LIN {X 0,Y 224.704,Z 635.837,A -85,B 0,C 180,E1 -21459.979,E2 -21459.979} C_VEL
LIN {X 0,Y 218.18,Z 645.105,A -85,B 0,C 180,E1 -21463.55,E2 -21463.55} C_VEL
LIN {X 0,Y 212.599,Z 652.771,A -85,B 0,C 180,E1 -21467.337,E2 -21467.337} C_VEL
LIN {X 0,Y 208.284,Z 658.451,A -85,B 0,C 180,E1 -21470.904,E2 -21470.904} C_VEL
LIN {X 0,Y 204.923,Z 662.804,A -85,B 0,C 180,E1 -21474.336,E2 -21474.336} C_VEL
LIN {X 0,Y 201.755,Z 666.821,A -85,B 0,C 180,E1 -21478.499,E2 -21478.499} C_VEL
LIN {X 0,Y 199.518,Z 669.692,A -85,B 0,C 180,E1 -21482.746,E2 -21482.746} C_VEL
LIN {X 0,Y 197.956,Z 671.64,A -85,B 0,C 180,E1 -21487.383,E2 -21487.383} C_VEL
LIN {X 0,Y 197.23,Z 672.274,A -85,B 0,C 180,E1 -21491.294,E2 -21491.294} C_VEL
LIN {X 0,Y 196.985,Z 672.087,A -85,B 0,C 180,E1 -21495.537,E2 -21495.537} C_VEL
LIN {X 0,Y 196.96,Z 670.835,A -85,B 0,C 180,E1 -21499.722,E2 -21499.722} C_VEL
LIN {X 0,Y 197.621,Z 668.047,A -85,B 0,C 180,E1 -21504.738,E2 -21504.738} C_VEL
LIN {X 0,Y 198.077,Z 665.462,A -85,B 0,C 180,E1 -21507.966,E2 -21507.966} C_VEL
LIN {X 0,Y 199.268,Z 661.253,A -85,B 0,C 180,E1 -21512.021,E2 -21512.021} C_VEL
LIN {X 0,Y 201.021,Z 655.948,A -85,B 0,C 180,E1 -21516.02,E2 -21516.02} C_VEL
LIN {X 0,Y 203.624,Z 649.403,A -85,B 0,C 180,E1 -21519.937,E2 -21519.937} C_VEL
LIN {X 0,Y 206.969,Z 641.573,A -85,B 0,C 180,E1 -21523.75,E2 -21523.75} C_VEL
LIN {X 0,Y 211.157,Z 632.216,A -85,B 0,C 180,E1 -21527.43,E2 -21527.43} C_VEL
LIN {X 0,Y 215.924,Z 621.042,A -85,B 0,C 180,E1 -21530.979,E2 -21530.979} C_VEL
LIN {X 0,Y 220.656,Z 609.454,A -85,B 0,C 180,E1 -21533.959,E2 -21533.959} C_VEL
LIN {X 0,Y 225.409,Z 596.841,A -85,B 0,C 180,E1 -21536.628,E2 -21536.628} C_VEL
LIN {X 0,Y 230.179,Z 583.089,A -85,B 0,C 180,E1 -21538.993,E2 -21538.993} C_VEL
LIN {X 0,Y 234.489,Z 569.519,A -85,B 0,C 180,E1 -21540.881,E2 -21540.881} C_VEL
LIN {X 0,Y 238.368,Z 554.82,A -85,B 0,C 180,E1 -21542.553,E2 -21542.553} C_VEL
LIN {X 0,Y 241.83,Z 539.767,A -85,B 0,C 180,E1 -21543.891,E2 -21543.891} C_VEL
LIN {X 0,Y 244.962,Z 523.135,A -85,B 0,C 180,E1 -21545.016,E2 -21545.016} C_VEL
LIN {X 0,Y 247.354,Z 506.595,A -85,B 0,C 180,E1 -21545.812,E2 -21545.812} C_VEL
LIN {X 0,Y 248.927,Z 489.58,A -85,B 0,C 180,E1 -21546.363,E2 -21546.363} C_VEL
LIN {X 0,Y 255.202,Z 390.664,A -85,B 0,C 180,E1 -21548.897,E2 -21548.897} C_VEL
LIN {X 0,Y 247.991,Z 376.871,A -85,B 0,C 180,E1 -21551.304,E2 -21551.304} C_VEL
LIN {X 0,Y 240.547,Z 364.083,A -85,B 0,C 180,E1 -21554.004,E2 -21554.004} C_VEL
LIN {X 0,Y 233.352,Z 353.034,A -85,B 0,C 180,E1 -21556.877,E2 -21556.877} C_VEL
LIN {X 0,Y 227.132,Z 344.318,A -85,B 0,C 180,E1 -21559.64,E2 -21559.64} C_VEL
LIN {X 0,Y 224.214,Z 340.378,A -85,B 0,C 180,E1 -21561.054,E2 -21561.054} C_VEL
LIN {X 0,Y 220.981,Z 336.041,A -85,B 0,C 180,E1 -21562.732,E2 -21562.732} C_VEL
LIN {X 0,Y 217.624,Z 331.577,A -85,B 0,C 180,E1 -21564.617,E2 -21564.617} C_VEL
LIN {X 0,Y 214.933,Z 328.464,A -85,B 0,C 180,E1 -21566.228,E2 -21566.228} C_VEL
LIN {X 0,Y 213.999,Z 326.917,A -85,B 0,C 180,E1 -21566.854,E2 -21566.854} C_VEL
LIN {X 0,Y 211.261,Z 324.389,A -85,B 0,C 180,E1 -21568.646,E2 -21568.646} C_VEL
LIN {X 0,Y 209.46,Z 321.523,A -85,B 0,C 180,E1 -21570.03,E2 -21570.03} C_VEL
LIN {X 0,Y 206.617,Z 319.284,A -85,B 0,C 180,E1 -21572.205,E2 -21572.205} C_VEL
LIN {X 0,Y 205.081,Z 316.402,A -85,B 0,C 180,E1 -21573.68,E2 -21573.68} C_VEL
LIN {X 0,Y 204.71,Z 315.862,A -85,B 0,C 180,E1 -21574.04,E2 -21574.04} C_VEL
LIN {X 0,Y 201.778,Z 314.105,A -85,B 0,C 180,E1 -21576.883,E2 -21576.883} C_VEL
LIN {X 0,Y 200.084,Z 311.584,A -85,B 0,C 180,E1 -21579.031,E2 -21579.031} C_VEL
LIN {X 0,Y 199.696,Z 309.917,A -85,B 0,C 180,E1 -21579.796,E2 -21579.796} C_VEL
LIN {X 0,Y 199.771,Z 309.895,A -85,B 0,C 180,E1 -21583.653,E2 -21583.653} C_VEL
LIN {X 0,Y 199.871,Z 309.874,A -85,B 0,C 180,E1 -21587.819,E2 -21587.819} C_VEL
LIN {X 0,Y 200.086,Z 309.867,A -85,B 0,C 180,E1 -21591.922,E2 -21591.922} C_VEL
LIN {X 0,Y 200.315,Z 309.84,A -85,B 0,C 180,E1 -21597.988,E2 -21597.988} C_VEL
LIN {X 0,Y 200.476,Z 309.798,A -85,B 0,C 180,E1 -21599.999,E2 -21599.999} C_VEL
LIN {X 0,Y 200.026,Z 309.876,A -85,B 0,C 180,E1 -21604.028,E2 -21604.028} C_VEL
LIN {X 0,Y 200.061,Z 309.893,A -85,B 0,C 180,E1 -21607.315,E2 -21607.315} C_VEL
LIN {X 0,Y 200.946,Z 312.488,A -85,B 0,C 180,E1 -21608.674,E2 -21608.674} C_VEL
LIN {X 0,Y 203.236,Z 315.062,A -85,B 0,C 180,E1 -21611.215,E2 -21611.215} C_VEL
LIN {X 0,Y 205.117,Z 316.12,A -85,B 0,C 180,E1 -21612.93,E2 -21612.93} C_VEL
LIN {X 0,Y 206.498,Z 318.89,A -85,B 0,C 180,E1 -21614.284,E2 -21614.284} C_VEL
LIN {X 0,Y 208.777,Z 321.042,A -85,B 0,C 180,E1 -21616.097,E2 -21616.097} C_VEL
LIN {X 0,Y 209.862,Z 321.847,A -85,B 0,C 180,E1 -21616.88,E2 -21616.88} C_VEL
LIN {X 0,Y 210.233,Z 322.642,A -85,B 0,C 180,E1 -21617.184,E2 -21617.184} C_VEL
LIN {X 0,Y 212.25,Z 327.471,A -85,B 0,C 180,E1 -21618.802,E2 -21618.802} C_VEL
LIN {X 0,Y 216.82,Z 339.371,A -85,B 0,C 180,E1 -21622.139,E2 -21622.139} C_VEL
LIN {X 0,Y 218.895,Z 342.438,A -85,B 0,C 180,E1 -21623.347,E2 -21623.347} C_VEL
LIN {X 0,Y 224.048,Z 349.555,A -85,B 0,C 180,E1 -21626.049,E2 -21626.049} C_VEL
LIN {X 0,Y 231.097,Z 359.699,A -85,B 0,C 180,E1 -21629.302,E2 -21629.302} C_VEL
LIN {X 0,Y 235.181,Z 366.487,A -85,B 0,C 180,E1 -21631.045,E2 -21631.045} C_VEL
LIN {X 0,Y 240.195,Z 376.25,A -85,B 0,C 180,E1 -21633.083,E2 -21633.083} C_VEL
LIN {X 0,Y 245.695,Z 387.89,A -85,B 0,C 180,E1 -21635.177,E2 -21635.177} C_VEL
LIN {X 0,Y 250.053,Z 398.361,A -85,B 0,C 180,E1 -21636.771,E2 -21636.771} C_VEL
LIN {X 0,Y 242.749,Z 508.587,A -85,B 0,C 180,E1 -21639.663,E2 -21639.663} C_VEL
LIN {X 0,Y 240.64,Z 525.362,A -85,B 0,C 180,E1 -21640.335,E2 -21640.335} C_VEL
LIN {X 0,Y 237.748,Z 541.464,A -85,B 0,C 180,E1 -21641.241,E2 -21641.241} C_VEL
LIN {X 0,Y 234.346,Z 556.741,A -85,B 0,C 180,E1 -21642.396,E2 -21642.396} C_VEL
LIN {X 0,Y 230.362,Z 571.885,A -85,B 0,C 180,E1 -21643.883,E2 -21643.883} C_VEL
LIN {X 0,Y 225.648,Z 586.645,A -85,B 0,C 180,E1 -21645.694,E2 -21645.694} C_VEL
LIN {X 0,Y 220.975,Z 600.129,A -85,B 0,C 180,E1 -21647.789,E2 -21647.789} C_VEL
LIN {X 0,Y 216.272,Z 612.309,A -85,B 0,C 180,E1 -21650.074,E2 -21650.074} C_VEL
LIN {X 0,Y 211.517,Z 623.913,A -85,B 0,C 180,E1 -21652.732,E2 -21652.732} C_VEL
LIN {X 0,Y 206.703,Z 635.08,A -85,B 0,C 180,E1 -21655.875,E2 -21655.875} C_VEL
LIN {X 0,Y 202.378,Z 644.779,A -85,B 0,C 180,E1 -21659.188,E2 -21659.188} C_VEL
LIN {X 0,Y 198.341,Z 654.189,A -85,B 0,C 180,E1 -21663.142,E2 -21663.142} C_VEL
LIN {X 0,Y 194.763,Z 662.887,A -85,B 0,C 180,E1 -21667.735,E2 -21667.735} C_VEL
LIN {X 0,Y 192.402,Z 669.547,A -85,B 0,C 180,E1 -21672.22,E2 -21672.22} C_VEL
LIN {X 0,Y 191.102,Z 674.172,A -85,B 0,C 180,E1 -21676.17,E2 -21676.17} C_VEL
LIN {X 0,Y 190.231,Z 678.879,A -85,B 0,C 180,E1 -21681.502,E2 -21681.502} C_VEL
LIN {X 0,Y 190.191,Z 681.456,A -85,B 0,C 180,E1 -21685.762,E2 -21685.762} C_VEL
LIN {X 0,Y 190.296,Z 682.962,A -85,B 0,C 180,E1 -21690,E2 -21690} C_VEL
LIN {X 0,Y 190.133,Z 683.504,A -85,B 0,C 180,E1 -21694.24,E2 -21694.24} C_VEL
LIN {X 0,Y 190.218,Z 683.045,A -85,B 0,C 180,E1 -21698.499,E2 -21698.499} C_VEL
LIN {X 0,Y 190.881,Z 681.67,A -85,B 0,C 180,E1 -21702.763,E2 -21702.763} C_VEL
LIN {X 0,Y 192.373,Z 679.322,A -85,B 0,C 180,E1 -21706.994,E2 -21706.994} C_VEL
LIN {X 0,Y 194.698,Z 676.014,A -85,B 0,C 180,E1 -21711.16,E2 -21711.16} C_VEL
LIN {X 0,Y 197.894,Z 671.662,A -85,B 0,C 180,E1 -21715.225,E2 -21715.225} C_VEL
LIN {X 0,Y 201.988,Z 666.267,A -85,B 0,C 180,E1 -21719.152,E2 -21719.152} C_VEL
LIN {X 0,Y 207.01,Z 659.627,A -85,B 0,C 180,E1 -21722.902,E2 -21722.902} C_VEL
LIN {X 0,Y 213.655,Z 650.625,A -85,B 0,C 180,E1 -21726.893,E2 -21726.893} C_VEL
LIN {X 0,Y 220.364,Z 641.039,A -85,B 0,C 180,E1 -21730.228,E2 -21730.228} C_VEL
LIN {X 0,Y 227.8,Z 629.661,A -85,B 0,C 180,E1 -21733.35,E2 -21733.35} C_VEL
LIN {X 0,Y 234.942,Z 617.871,A -85,B 0,C 180,E1 -21735.884,E2 -21735.884} C_VEL
LIN {X 0,Y 241.451,Z 605.863,A -85,B 0,C 180,E1 -21737.975,E2 -21737.975} C_VEL
LIN {X 0,Y 248.161,Z 592.197,A -85,B 0,C 180,E1 -21739.876,E2 -21739.876} C_VEL
LIN {X 0,Y 254.139,Z 578.552,A -85,B 0,C 180,E1 -21741.374,E2 -21741.374} C_VEL
LIN {X 0,Y 259.557,Z 563.781,A -85,B 0,C 180,E1 -21742.692,E2 -21742.692} C_VEL
LIN {X 0,Y 264.238,Z 548.652,A -85,B 0,C 180,E1 -21743.729,E2 -21743.729} C_VEL
LIN {X 0,Y 268.405,Z 531.917,A -85,B 0,C 180,E1 -21744.591,E2 -21744.591} C_VEL
LIN {X 0,Y 271.417,Z 515.904,A -85,B 0,C 180,E1 -21745.177,E2 -21745.177} C_VEL
LIN {X 0,Y 273.367,Z 498.876,A -85,B 0,C 180,E1 -21745.66,E2 -21745.66} C_VEL
LIN {X 0,Y 279.986,Z 417.951,A -85,B 0,C 180,E1 -21747.514,E2 -21747.514} C_VEL
LIN {X 0,Y 275.543,Z 408.438,A -85,B 0,C 180,E1 -21749.967,E2 -21749.967} C_VEL
LIN {X 0,Y 271.529,Z 400.291,A -85,B 0,C 180,E1 -21752.452,E2 -21752.452} C_VEL
LIN {X 0,Y 266.969,Z 391.871,A -85,B 0,C 180,E1 -21755.707,E2 -21755.707} C_VEL
LIN {X 0,Y 263.419,Z 386.396,A -85,B 0,C 180,E1 -21758.705,E2 -21758.705} C_VEL
LIN {X 0,Y 260.513,Z 382.099,A -85,B 0,C 180,E1 -21761.74,E2 -21761.74} C_VEL
LIN {X 0,Y 258.214,Z 378.675,A -85,B 0,C 180,E1 -21764.965,E2 -21764.965} C_VEL
LIN {X 0,Y 257.777,Z 377.656,A -85,B 0,C 180,E1 -21765.797,E2 -21765.797} C_VEL
LIN {X 0,Y 255.553,Z 374.982,A -85,B 0,C 180,E1 -21773.018,E2 -21773.018} C_VEL
LIN {X 0,Y 256.078,Z 375.739,A -85,B 0,C 180,E1 -21777.641,E2 -21777.641} C_VEL
LIN {X 0,Y 258.062,Z 377.883,A -85,B 0,C 180,E1 -21782.12,E2 -21782.12} C_VEL
LIN {X 0,Y 260.464,Z 381.798,A -85,B 0,C 180,E1 -21785.614,E2 -21785.614} C_VEL
LIN {X 0,Y 261.202,Z 382.927,A -85,B 0,C 180,E1 -21786.47,E2 -21786.47} C_VEL
LIN {X 0,Y 264.003,Z 387.156,A -85,B 0,C 180,E1 -21789.264,E2 -21789.264} C_VEL
LIN {X 0,Y 267.122,Z 392.052,A -85,B 0,C 180,E1 -21791.85,E2 -21791.85} C_VEL
LIN {X 0,Y 271.202,Z 398.501,A -85,B 0,C 180,E1 -21794.696,E2 -21794.696} C_VEL
LIN {X 0,Y 276.177,Z 406.975,A -85,B 0,C 180,E1 -21797.674,E2 -21797.674} C_VEL
LIN {X 0,Y 280.247,Z 414.31,A -85,B 0,C 180,E1 -21799.832,E2 -21799.832} C_VEL
LIN {X 0,Y 273.006,Z 500.411,A -85,B 0,C 180,E1 -21801.818,E2 -21801.818} C_VEL
LIN {X 0,Y 270.274,Z 517.579,A -85,B 0,C 180,E1 -21802.37,E2 -21802.37} C_VEL
LIN {X 0,Y 266.884,Z 533.687,A -85,B 0,C 180,E1 -21803.19,E2 -21803.19} C_VEL
LIN {X 0,Y 262.691,Z 548.993,A -85,B 0,C 180,E1 -21804.19,E2 -21804.19} C_VEL
LIN {X 0,Y 257.769,Z 563.8,A -85,B 0,C 180,E1 -21805.425,E2 -21805.425} C_VEL
LIN {X 0,Y 252.193,Z 577.919,A -85,B 0,C 180,E1 -21806.904,E2 -21806.904} C_VEL
LIN {X 0,Y 245.781,Z 591.955,A -85,B 0,C 180,E1 -21808.756,E2 -21808.756} C_VEL
LIN {X 0,Y 239.278,Z 604.411,A -85,B 0,C 180,E1 -21810.782,E2 -21810.782} C_VEL
LIN {X 0,Y 232.265,Z 616.607,A -85,B 0,C 180,E1 -21813.266,E2 -21813.266} C_VEL
LIN {X 0,Y 225.616,Z 627.114,A -85,B 0,C 180,E1 -21815.913,E2 -21815.913} C_VEL
LIN {X 0,Y 219.013,Z 636.625,A -85,B 0,C 180,E1 -21818.906,E2 -21818.906} C_VEL
LIN {X 0,Y 212.212,Z 645.786,A -85,B 0,C 180,E1 -21822.534,E2 -21822.534} C_VEL
LIN {X 0,Y 206.881,Z 652.722,A -85,B 0,C 180,E1 -21826.022,E2 -21826.022} C_VEL
LIN {X 0,Y 201.943,Z 658.863,A -85,B 0,C 180,E1 -21829.966,E2 -21829.966} C_VEL
LIN {X 0,Y 197.855,Z 663.805,A -85,B 0,C 180,E1 -21834.121,E2 -21834.121} C_VEL
LIN {X 0,Y 195.325,Z 666.777,A -85,B 0,C 180,E1 -21837.335,E2 -21837.335} C_VEL
LIN {X 0,Y 192.83,Z 669.746,A -85,B 0,C 180,E1 -21841.718,E2 -21841.718} C_VEL
LIN {X 0,Y 191.144,Z 671.643,A -85,B 0,C 180,E1 -21846.143,E2 -21846.143} C_VEL
LIN {X 0,Y 190.213,Z 672.467,A -85,B 0,C 180,E1 -21850.577,E2 -21850.577} C_VEL
LIN {X 0,Y 189.912,Z 672.341,A -85,B 0,C 180,E1 -21854.986,E2 -21854.986} C_VEL
LIN {X 0,Y 189.838,Z 671.158,A -85,B 0,C 180,E1 -21859.332,E2 -21859.332} C_VEL
LIN {X 0,Y 190.282,Z 669.078,A -85,B 0,C 180,E1 -21863.638,E2 -21863.638} C_VEL
LIN {X 0,Y 190.973,Z 665.916,A -85,B 0,C 180,E1 -21867.891,E2 -21867.891} C_VEL
LIN {X 0,Y 192.18,Z 661.802,A -85,B 0,C 180,E1 -21872.096,E2 -21872.096} C_VEL
LIN {X 0,Y 193.97,Z 656.546,A -85,B 0,C 180,E1 -21876.24,E2 -21876.24} C_VEL
LIN {X 0,Y 196.647,Z 650.108,A -85,B 0,C 180,E1 -21880.294,E2 -21880.294} C_VEL
LIN {X 0,Y 200.106,Z 642.393,A -85,B 0,C 180,E1 -21884.232,E2 -21884.232} C_VEL
LIN {X 0,Y 204.419,Z 633.103,A -85,B 0,C 180,E1 -21888.024,E2 -21888.024} C_VEL
LIN {X 0,Y 208.705,Z 623.53,A -85,B 0,C 180,E1 -21891.223,E2 -21891.223} C_VEL
LIN {X 0,Y 213.549,Z 612.39,A -85,B 0,C 180,E1 -21894.291,E2 -21894.291} C_VEL
LIN {X 0,Y 218.336,Z 600.324,A -85,B 0,C 180,E1 -21897.043,E2 -21897.043} C_VEL
LIN {X 0,Y 223.623,Z 585.949,A -85,B 0,C 180,E1 -21899.669,E2 -21899.669} C_VEL
LIN {X 0,Y 228.502,Z 571.289,A -85,B 0,C 180,E1 -21901.783,E2 -21901.783} C_VEL
LIN {X 0,Y 232.522,Z 556.903,A -85,B 0,C 180,E1 -21903.477,E2 -21903.477} C_VEL
LIN {X 0,Y 236.289,Z 541.265,A -85,B 0,C 180,E1 -21904.929,E2 -21904.929} C_VEL
LIN {X 0,Y 239.548,Z 525.061,A -85,B 0,C 180,E1 -21906.058,E2 -21906.058} C_VEL
LIN {X 0,Y 241.952,Z 509.331,A -85,B 0,C 180,E1 -21906.87,E2 -21906.87} C_VEL
LIN {X 0,Y 243.738,Z 491.917,A -85,B 0,C 180,E1 -21907.458,E2 -21907.458} C_VEL
LIN {X 0,Y 250.218,Z 393.361,A -85,B 0,C 180,E1 -21910.013,E2 -21910.013} C_VEL
LIN {X 0,Y 243.332,Z 380.216,A -85,B 0,C 180,E1 -21912.435,E2 -21912.435} C_VEL
LIN {X 0,Y 236.792,Z 368.826,A -85,B 0,C 180,E1 -21914.936,E2 -21914.936} C_VEL
LIN {X 0,Y 230.444,Z 358.854,A -85,B 0,C 180,E1 -21917.587,E2 -21917.587} C_VEL
LIN {X 0,Y 224.274,Z 350.024,A -85,B 0,C 180,E1 -21920.446,E2 -21920.446} C_VEL
LIN {X 0,Y 221.012,Z 345.557,A -85,B 0,C 180,E1 -21922.106,E2 -21922.106} C_VEL
LIN {X 0,Y 218.342,Z 341.865,A -85,B 0,C 180,E1 -21923.567,E2 -21923.567} C_VEL
LIN {X 0,Y 215.202,Z 337.669,A -85,B 0,C 180,E1 -21925.411,E2 -21925.411} C_VEL
LIN {X 0,Y 212.429,Z 334.12,A -85,B 0,C 180,E1 -21927.178,E2 -21927.178} C_VEL
LIN {X 0,Y 210.816,Z 332.472,A -85,B 0,C 180,E1 -21928.25,E2 -21928.25} C_VEL
LIN {X 0,Y 208.297,Z 329.149,A -85,B 0,C 180,E1 -21930.119,E2 -21930.119} C_VEL
LIN {X 0,Y 207.591,Z 328.144,A -85,B 0,C 180,E1 -21930.681,E2 -21930.681} C_VEL
LIN {X 0,Y 204.877,Z 325.744,A -85,B 0,C 180,E1 -21932.871,E2 -21932.871} C_VEL
LIN {X 0,Y 203.357,Z 322.849,A -85,B 0,C 180,E1 -21934.404,E2 -21934.404} C_VEL
LIN {X 0,Y 200.049,Z 320.467,A -85,B 0,C 180,E1 -21937.81,E2 -21937.81} C_VEL
LIN {X 0,Y 198.536,Z 317.752,A -85,B 0,C 180,E1 -21939.943,E2 -21939.943} C_VEL
LIN {X 0,Y 198.159,Z 316.828,A -85,B 0,C 180,E1 -21940.578,E2 -21940.578} C_VEL
LIN {X 0,Y 194.367,Z 314.325,A -85,B 0,C 180,E1 -21948.528,E2 -21948.528} C_VEL
LIN {X 0,Y 193.907,Z 313.392,A -85,B 0,C 180,E1 -21951.663,E2 -21951.663} C_VEL
LIN {X 0,Y 194.521,Z 313.913,A -85,B 0,C 180,E1 -21958.446,E2 -21958.446} C_VEL
LIN {X 0,Y 195.475,Z 314.975,A -85,B 0,C 180,E1 -21961.286,E2 -21961.286} C_VEL
LIN {X 0,Y 197.619,Z 316.548,A -85,B 0,C 180,E1 -21965.271,E2 -21965.271} C_VEL
LIN {X 0,Y 198.722,Z 316.968,A -85,B 0,C 180,E1 -21966.79,E2 -21966.79} C_VEL
LIN {X 0,Y 199.805,Z 319.573,A -85,B 0,C 180,E1 -21968.426,E2 -21968.426} C_VEL
LIN {X 0,Y 202.055,Z 322.006,A -85,B 0,C 180,E1 -21970.964,E2 -21970.964} C_VEL
LIN {X 0,Y 203.513,Z 322.95,A -85,B 0,C 180,E1 -21972.349,E2 -21972.349} C_VEL
LIN {X 0,Y 205.331,Z 326.072,A -85,B 0,C 180,E1 -21974.122,E2 -21974.122} C_VEL
LIN {X 0,Y 208.079,Z 328.6,A -85,B 0,C 180,E1 -21976.309,E2 -21976.309} C_VEL
LIN {X 0,Y 210.43,Z 332.062,A -85,B 0,C 180,E1 -21978.096,E2 -21978.096} C_VEL
LIN {X 0,Y 212.297,Z 333.845,A -85,B 0,C 180,E1 -21979.331,E2 -21979.331} C_VEL
LIN {X 0,Y 214.989,Z 337.505,A -85,B 0,C 180,E1 -21981.074,E2 -21981.074} C_VEL
LIN {X 0,Y 216.463,Z 339.261,A -85,B 0,C 180,E1 -21981.954,E2 -21981.954} C_VEL
LIN {X 0,Y 218.895,Z 342.438,A -85,B 0,C 180,E1 -21983.347,E2 -21983.347} C_VEL
LIN {X 0,Y 220.304,Z 344.535,A -85,B 0,C 180,E1 -21984.13,E2 -21984.13} C_VEL
LIN {X 0,Y 221.475,Z 347.199,A -85,B 0,C 180,E1 -21984.818,E2 -21984.818} C_VEL
LIN {X 0,Y 225.862,Z 361.333,A -85,B 0,C 180,E1 -21987.461,E2 -21987.461} C_VEL
LIN {X 0,Y 228.001,Z 365.171,A -85,B 0,C 180,E1 -21988.481,E2 -21988.481} C_VEL
LIN {X 0,Y 231.897,Z 371.817,A -85,B 0,C 180,E1 -21990.222,E2 -21990.222} C_VEL
LIN {X 0,Y 236.874,Z 381.772,A -85,B 0,C 180,E1 -21992.342,E2 -21992.342} C_VEL
LIN {X 0,Y 242.247,Z 393.639,A -85,B 0,C 180,E1 -21994.483,E2 -21994.483} C_VEL
LIN {X 0,Y 245.234,Z 400.816,A -85,B 0,C 180,E1 -21995.625,E2 -21995.625} C_VEL
LIN {X 0,Y 237.721,Z 509.196,A -85,B 0,C 180,E1 -21998.478,E2 -21998.478} C_VEL
LIN {X 0,Y 235.469,Z 526.323,A -85,B 0,C 180,E1 -21999.188,E2 -21999.188} C_VEL
LIN {X 0,Y 232.505,Z 541.938,A -85,B 0,C 180,E1 -22000.082,E2 -22000.082} C_VEL
LIN {X 0,Y 228.731,Z 558.063,A -85,B 0,C 180,E1 -22001.335,E2 -22001.335} C_VEL
LIN {X 0,Y 224.903,Z 572.108,A -85,B 0,C 180,E1 -22002.748,E2 -22002.748} C_VEL
LIN {X 0,Y 220.172,Z 586.443,A -85,B 0,C 180,E1 -22004.529,E2 -22004.529} C_VEL
LIN {X 0,Y 215.218,Z 600.232,A -85,B 0,C 180,E1 -22006.705,E2 -22006.705} C_VEL
LIN {X 0,Y 209.912,Z 613.358,A -85,B 0,C 180,E1 -22009.242,E2 -22009.242} C_VEL
LIN {X 0,Y 204.673,Z 625.551,A -85,B 0,C 180,E1 -22012.162,E2 -22012.162} C_VEL
LIN {X 0,Y 200.055,Z 635.84,A -85,B 0,C 180,E1 -22015.19,E2 -22015.19} C_VEL
LIN {X 0,Y 195.587,Z 645.376,A -85,B 0,C 180,E1 -22018.599,E2 -22018.599} C_VEL
LIN {X 0,Y 191.416,Z 654.642,A -85,B 0,C 180,E1 -22022.681,E2 -22022.681} C_VEL
LIN {X 0,Y 188.087,Z 662.381,A -85,B 0,C 180,E1 -22026.9,E2 -22026.9} C_VEL
LIN {X 0,Y 185.758,Z 668.434,A -85,B 0,C 180,E1 -22031.056,E2 -22031.056} C_VEL
LIN {X 0,Y 184.142,Z 673.77,A -85,B 0,C 180,E1 -22035.636,E2 -22035.636} C_VEL
LIN {X 0,Y 183.162,Z 678.54,A -85,B 0,C 180,E1 -22041.172,E2 -22041.172} C_VEL
LIN {X 0,Y 183.111,Z 681.148,A -85,B 0,C 180,E1 -22045.598,E2 -22045.598} C_VEL
LIN {X 0,Y 183.199,Z 682.712,A -85,B 0,C 180,E1 -22050,E2 -22050} C_VEL
LIN {X 0,Y 183.029,Z 683.281,A -85,B 0,C 180,E1 -22054.405,E2 -22054.405} C_VEL
LIN {X 0,Y 183.159,Z 682.879,A -85,B 0,C 180,E1 -22058.829,E2 -22058.829} C_VEL
LIN {X 0,Y 183.889,Z 681.531,A -85,B 0,C 180,E1 -22063.257,E2 -22063.257} C_VEL
LIN {X 0,Y 185.517,Z 679.244,A -85,B 0,C 180,E1 -22067.642,E2 -22067.642} C_VEL
LIN {X 0,Y 188.002,Z 675.97,A -85,B 0,C 180,E1 -22071.952,E2 -22071.952} C_VEL
LIN {X 0,Y 191.407,Z 671.682,A -85,B 0,C 180,E1 -22076.143,E2 -22076.143} C_VEL
LIN {X 0,Y 195.737,Z 666.321,A -85,B 0,C 180,E1 -22080.177,E2 -22080.177} C_VEL
LIN {X 0,Y 201.036,Z 659.752,A -85,B 0,C 180,E1 -22084.011,E2 -22084.011} C_VEL
LIN {X 0,Y 207.991,Z 650.829,A -85,B 0,C 180,E1 -22088.073,E2 -22088.073} C_VEL
LIN {X 0,Y 214.961,Z 641.341,A -85,B 0,C 180,E1 -22091.457,E2 -22091.457} C_VEL
LIN {X 0,Y 222.676,Z 630.062,A -85,B 0,C 180,E1 -22094.608,E2 -22094.608} C_VEL
LIN {X 0,Y 230.066,Z 618.339,A -85,B 0,C 180,E1 -22097.151,E2 -22097.151} C_VEL
LIN {X 0,Y 237.263,Z 605.581,A -85,B 0,C 180,E1 -22099.381,E2 -22099.381} C_VEL
LIN {X 0,Y 244.312,Z 591.685,A -85,B 0,C 180,E1 -22101.288,E2 -22101.288} C_VEL
LIN {X 0,Y 250.409,Z 577.981,A -85,B 0,C 180,E1 -22102.786,E2 -22102.786} C_VEL
LIN {X 0,Y 255.983,Z 563.171,A -85,B 0,C 180,E1 -22104.089,E2 -22104.089} C_VEL
LIN {X 0,Y 260.819,Z 547.936,A -85,B 0,C 180,E1 -22105.102,E2 -22105.102} C_VEL
LIN {X 0,Y 264.973,Z 531.469,A -85,B 0,C 180,E1 -22105.941,E2 -22105.941} C_VEL
LIN {X 0,Y 268.089,Z 515.106,A -85,B 0,C 180,E1 -22106.525,E2 -22106.525} C_VEL
LIN {X 0,Y 270.033,Z 498.486,A -85,B 0,C 180,E1 -22106.988,E2 -22106.988} C_VEL
LIN {X 0,Y 276.521,Z 421.533,A -85,B 0,C 180,E1 -22108.743,E2 -22108.743} C_VEL
LIN {X 0,Y 272.814,Z 413.288,A -85,B 0,C 180,E1 -22110.935,E2 -22110.935} C_VEL
LIN {X 0,Y 269.158,Z 405.674,A -85,B 0,C 180,E1 -22113.335,E2 -22113.335} C_VEL
LIN {X 0,Y 264.696,Z 397.181,A -85,B 0,C 180,E1 -22116.749,E2 -22116.749} C_VEL
LIN {X 0,Y 261.859,Z 392.902,A -85,B 0,C 180,E1 -22119.285,E2 -22119.285} C_VEL
LIN {X 0,Y 259.2,Z 388.803,A -85,B 0,C 180,E1 -22122.219,E2 -22122.219} C_VEL
LIN {X 0,Y 257.029,Z 385.312,A -85,B 0,C 180,E1 -22125.468,E2 -22125.468} C_VEL
LIN {X 0,Y 256.69,Z 384.609,A -85,B 0,C 180,E1 -22126.134,E2 -22126.134} C_VEL
LIN {X 0,Y 254.678,Z 382.039,A -85,B 0,C 180,E1 -22132.994,E2 -22132.994} C_VEL
LIN {X 0,Y 255.195,Z 382.804,A -85,B 0,C 180,E1 -22137.633,E2 -22137.633} C_VEL
LIN {X 0,Y 257.006,Z 384.816,A -85,B 0,C 180,E1 -22141.848,E2 -22141.848} C_VEL
LIN {X 0,Y 259.246,Z 388.619,A -85,B 0,C 180,E1 -22145.25,E2 -22145.25} C_VEL
LIN {X 0,Y 259.932,Z 389.743,A -85,B 0,C 180,E1 -22146.088,E2 -22146.088} C_VEL
LIN {X 0,Y 262.662,Z 393.994,A -85,B 0,C 180,E1 -22148.912,E2 -22148.912} C_VEL
LIN {X 0,Y 265.602,Z 398.724,A -85,B 0,C 180,E1 -22151.435,E2 -22151.435} C_VEL
LIN {X 0,Y 269.369,Z 404.957,A -85,B 0,C 180,E1 -22154.174,E2 -22154.174} C_VEL
LIN {X 0,Y 273.813,Z 412.705,A -85,B 0,C 180,E1 -22156.946,E2 -22156.946} C_VEL
LIN {X 0,Y 276.752,Z 418.174,A -85,B 0,C 180,E1 -22158.602,E2 -22158.602} C_VEL
LIN {X 0,Y 269.648,Z 500.46,A -85,B 0,C 180,E1 -22160.501,E2 -22160.501} C_VEL
LIN {X 0,Y 266.851,Z 517.656,A -85,B 0,C 180,E1 -22161.042,E2 -22161.042} C_VEL
LIN {X 0,Y 263.514,Z 533.239,A -85,B 0,C 180,E1 -22161.829,E2 -22161.829} C_VEL
LIN {X 0,Y 258.884,Z 549.638,A -85,B 0,C 180,E1 -22162.881,E2 -22162.881} C_VEL
LIN {X 0,Y 253.52,Z 565.155,A -85,B 0,C 180,E1 -22164.189,E2 -22164.189} C_VEL
LIN {X 0,Y 247.642,Z 579.482,A -85,B 0,C 180,E1 -22165.702,E2 -22165.702} C_VEL
LIN {X 0,Y 240.829,Z 593.763,A -85,B 0,C 180,E1 -22167.619,E2 -22167.619} C_VEL
LIN {X 0,Y 233.771,Z 606.582,A -85,B 0,C 180,E1 -22169.762,E2 -22169.762} C_VEL
LIN {X 0,Y 227.174,Z 617.534,A -85,B 0,C 180,E1 -22172.063,E2 -22172.063} C_VEL
LIN {X 0,Y 220.531,Z 627.594,A -85,B 0,C 180,E1 -22174.627,E2 -22174.627} C_VEL
LIN {X 0,Y 213.396,Z 637.421,A -85,B 0,C 180,E1 -22177.775,E2 -22177.775} C_VEL
LIN {X 0,Y 207.167,Z 645.424,A -85,B 0,C 180,E1 -22180.99,E2 -22180.99} C_VEL
LIN {X 0,Y 201.197,Z 652.812,A -85,B 0,C 180,E1 -22184.726,E2 -22184.726} C_VEL
LIN {X 0,Y 195.019,Z 660.041,A -85,B 0,C 180,E1 -22189.558,E2 -22189.558} C_VEL
LIN {X 0,Y 190.416,Z 665.215,A -85,B 0,C 180,E1 -22194.293,E2 -22194.293} C_VEL
LIN {X 0,Y 186.473,Z 669.534,A -85,B 0,C 180,E1 -22200.097,E2 -22200.097} C_VEL
LIN {X 0,Y 184.32,Z 671.744,A -85,B 0,C 180,E1 -22205.202,E2 -22205.202} C_VEL
LIN {X 0,Y 183.218,Z 672.66,A -85,B 0,C 180,E1 -22209.804,E2 -22209.804} C_VEL
LIN {X 0,Y 182.832,Z 672.577,A -85,B 0,C 180,E1 -22214.39,E2 -22214.39} C_VEL
LIN {X 0,Y 182.719,Z 671.482,A -85,B 0,C 180,E1 -22218.912,E2 -22218.912} C_VEL
LIN {X 0,Y 183.127,Z 669.453,A -85,B 0,C 180,E1 -22223.388,E2 -22223.388} C_VEL
LIN {X 0,Y 183.524,Z 668.021,A -85,B 0,C 180,E1 -22225.607,E2 -22225.607} C_VEL
LIN {X 0,Y 184.751,Z 663.415,A -85,B 0,C 180,E1 -22231.09,E2 -22231.09} C_VEL
LIN {X 0,Y 186.398,Z 658.557,A -85,B 0,C 180,E1 -22235.409,E2 -22235.409} C_VEL
LIN {X 0,Y 188.941,Z 652.523,A -85,B 0,C 180,E1 -22239.636,E2 -22239.636} C_VEL
LIN {X 0,Y 192.789,Z 644.179,A -85,B 0,C 180,E1 -22244.245,E2 -22244.245} C_VEL
LIN {X 0,Y 197.078,Z 635.205,A -85,B 0,C 180,E1 -22248.182,E2 -22248.182} C_VEL
LIN {X 0,Y 201.49,Z 626.007,A -85,B 0,C 180,E1 -22251.484,E2 -22251.484} C_VEL
LIN {X 0,Y 206.424,Z 615.23,A -85,B 0,C 180,E1 -22254.649,E2 -22254.649} C_VEL
LIN {X 0,Y 210.885,Z 604.487,A -85,B 0,C 180,E1 -22257.273,E2 -22257.273} C_VEL
LIN {X 0,Y 215.807,Z 592.051,A -85,B 0,C 180,E1 -22259.777,E2 -22259.777} C_VEL
LIN {X 0,Y 220.718,Z 578.613,A -85,B 0,C 180,E1 -22261.962,E2 -22261.962} C_VEL
LIN {X 0,Y 225.357,Z 563.96,A -85,B 0,C 180,E1 -22263.88,E2 -22263.88} C_VEL
LIN {X 0,Y 229.157,Z 549.862,A -85,B 0,C 180,E1 -22265.371,E2 -22265.371} C_VEL
LIN {X 0,Y 232.385,Z 536.028,A -85,B 0,C 180,E1 -22266.541,E2 -22266.541} C_VEL
LIN {X 0,Y 235.594,Z 518.759,A -85,B 0,C 180,E1 -22267.633,E2 -22267.633} C_VEL
LIN {X 0,Y 237.885,Z 502.101,A -85,B 0,C 180,E1 -22268.346,E2 -22268.346} C_VEL
LIN {X 0,Y 239.831,Z 477.305,A -85,B 0,C 180,E1 -22269.052,E2 -22269.052} C_VEL
LIN {X 0,Y 245.314,Z 396.202,A -85,B 0,C 180,E1 -22271.17,E2 -22271.17} C_VEL
LIN {X 0,Y 238.598,Z 383.136,A -85,B 0,C 180,E1 -22273.681,E2 -22273.681} C_VEL
LIN {X 0,Y 231.532,Z 370.911,A -85,B 0,C 180,E1 -22276.564,E2 -22276.564} C_VEL
LIN {X 0,Y 224.888,Z 360.626,A -85,B 0,C 180,E1 -22279.574,E2 -22279.574} C_VEL
LIN {X 0,Y 219.205,Z 352.459,A -85,B 0,C 180,E1 -22282.47,E2 -22282.47} C_VEL
LIN {X 0,Y 215.709,Z 347.69,A -85,B 0,C 180,E1 -22284.442,E2 -22284.442} C_VEL
LIN {X 0,Y 213.092,Z 344.034,A -85,B 0,C 180,E1 -22286.056,E2 -22286.056} C_VEL
LIN {X 0,Y 210.209,Z 340.171,A -85,B 0,C 180,E1 -22287.985,E2 -22287.985} C_VEL
LIN {X 0,Y 206.875,Z 336.357,A -85,B 0,C 180,E1 -22290.419,E2 -22290.419} C_VEL
LIN {X 0,Y 205.941,Z 334.827,A -85,B 0,C 180,E1 -22291.201,E2 -22291.201} C_VEL
LIN {X 0,Y 203.332,Z 332.415,A -85,B 0,C 180,E1 -22293.391,E2 -22293.391} C_VEL
LIN {X 0,Y 201.759,Z 329.563,A -85,B 0,C 180,E1 -22295.026,E2 -22295.026} C_VEL
LIN {X 0,Y 198.699,Z 327.195,A -85,B 0,C 180,E1 -22298.334,E2 -22298.334} C_VEL
LIN {X 0,Y 197.14,Z 324.239,A -85,B 0,C 180,E1 -22300.677,E2 -22300.677} C_VEL
LIN {X 0,Y 196.783,Z 323.727,A -85,B 0,C 180,E1 -22301.249,E2 -22301.249} C_VEL
LIN {X 0,Y 193.212,Z 320.837,A -85,B 0,C 180,E1 -22310.005,E2 -22310.005} C_VEL
LIN {X 0,Y 193.035,Z 320.435,A -85,B 0,C 180,E1 -22311.625,E2 -22311.625} C_VEL
LIN {X 0,Y 193.638,Z 320.971,A -85,B 0,C 180,E1 -22318.439,E2 -22318.439} C_VEL
LIN {X 0,Y 196.628,Z 323.561,A -85,B 0,C 180,E1 -22325.125,E2 -22325.125} C_VEL
LIN {X 0,Y 197.431,Z 323.912,A -85,B 0,C 180,E1 -22326.277,E2 -22326.277} C_VEL
LIN {X 0,Y 198.773,Z 326.803,A -85,B 0,C 180,E1 -22328.313,E2 -22328.313} C_VEL
LIN {X 0,Y 201.182,Z 329.112,A -85,B 0,C 180,E1 -22331.013,E2 -22331.013} C_VEL
LIN {X 0,Y 201.945,Z 329.705,A -85,B 0,C 180,E1 -22331.765,E2 -22331.765} C_VEL
LIN {X 0,Y 203.822,Z 332.815,A -85,B 0,C 180,E1 -22333.648,E2 -22333.648} C_VEL
LIN {X 0,Y 206.335,Z 335.274,A -85,B 0,C 180,E1 -22335.732,E2 -22335.732} C_VEL
LIN {X 0,Y 208.878,Z 338.866,A -85,B 0,C 180,E1 -22337.713,E2 -22337.713} C_VEL
LIN {X 0,Y 210.331,Z 340.353,A -85,B 0,C 180,E1 -22338.712,E2 -22338.712} C_VEL
LIN {X 0,Y 213.324,Z 344.307,A -85,B 0,C 180,E1 -22340.694,E2 -22340.694} C_VEL
LIN {X 0,Y 217.813,Z 350.43,A -85,B 0,C 180,E1 -22343.374,E2 -22343.374} C_VEL
LIN {X 0,Y 223.048,Z 357.81,A -85,B 0,C 180,E1 -22346.135,E2 -22346.135} C_VEL
LIN {X 0,Y 228.001,Z 365.171,A -85,B 0,C 180,E1 -22348.481,E2 -22348.481} C_VEL
LIN {X 0,Y 229.466,Z 367.623,A -85,B 0,C 180,E1 -22349.146,E2 -22349.146} C_VEL
LIN {X 0,Y 231.071,Z 372.26,A -85,B 0,C 180,E1 -22349.957,E2 -22349.957} C_VEL
LIN {X 0,Y 234.396,Z 388.309,A -85,B 0,C 180,E1 -22351.886,E2 -22351.886} C_VEL
LIN {X 0,Y 235.531,Z 391.563,A -85,B 0,C 180,E1 -22352.404,E2 -22352.404} C_VEL
LIN {X 0,Y 240.447,Z 403.254,A -85,B 0,C 180,E1 -22354.416,E2 -22354.416} C_VEL
LIN {X 0,Y 232.936,Z 508.277,A -85,B 0,C 180,E1 -22357.196,E2 -22357.196} C_VEL
LIN {X 0,Y 230.678,Z 525.206,A -85,B 0,C 180,E1 -22357.882,E2 -22357.882} C_VEL
LIN {X 0,Y 227.642,Z 541.089,A -85,B 0,C 180,E1 -22358.781,E2 -22358.781} C_VEL
LIN {X 0,Y 224.029,Z 556.355,A -85,B 0,C 180,E1 -22359.948,E2 -22359.948} C_VEL
LIN {X 0,Y 220.069,Z 570.614,A -85,B 0,C 180,E1 -22361.368,E2 -22361.368} C_VEL
LIN {X 0,Y 215.321,Z 584.674,A -85,B 0,C 180,E1 -22363.089,E2 -22363.089} C_VEL
LIN {X 0,Y 210.002,Z 599.133,A -85,B 0,C 180,E1 -22365.349,E2 -22365.349} C_VEL
LIN {X 0,Y 204.473,Z 612.408,A -85,B 0,C 180,E1 -22367.915,E2 -22367.915} C_VEL
LIN {X 0,Y 199.436,Z 623.788,A -85,B 0,C 180,E1 -22370.632,E2 -22370.632} C_VEL
LIN {X 0,Y 194.154,Z 635.068,A -85,B 0,C 180,E1 -22373.969,E2 -22373.969} C_VEL
LIN {X 0,Y 189.431,Z 644.699,A -85,B 0,C 180,E1 -22377.455,E2 -22377.455} C_VEL
LIN {X 0,Y 185.026,Z 654.054,A -85,B 0,C 180,E1 -22381.654,E2 -22381.654} C_VEL
LIN {X 0,Y 181.455,Z 661.848,A -85,B 0,C 180,E1 -22386.004,E2 -22386.004} C_VEL
LIN {X 0,Y 178.369,Z 669.645,A -85,B 0,C 180,E1 -22391.627,E2 -22391.627} C_VEL
LIN {X 0,Y 176.842,Z 674.455,A -85,B 0,C 180,E1 -22396.205,E2 -22396.205} C_VEL
LIN {X 0,Y 176.082,Z 678.199,A -85,B 0,C 180,E1 -22400.813,E2 -22400.813} C_VEL
LIN {X 0,Y 176.015,Z 680.84,A -85,B 0,C 180,E1 -22405.42,E2 -22405.42} C_VEL
LIN {X 0,Y 176.104,Z 682.461,A -85,B 0,C 180,E1 -22410,E2 -22410} C_VEL
LIN {X 0,Y 175.935,Z 683.058,A -85,B 0,C 180,E1 -22414.583,E2 -22414.583} C_VEL
LIN {X 0,Y 176.085,Z 682.713,A -85,B 0,C 180,E1 -22419.187,E2 -22419.187} C_VEL
LIN {X 0,Y 176.914,Z 681.395,A -85,B 0,C 180,E1 -22423.79,E2 -22423.79} C_VEL
LIN {X 0,Y 178.695,Z 679.169,A -85,B 0,C 180,E1 -22428.339,E2 -22428.339} C_VEL
LIN {X 0,Y 181.345,Z 675.925,A -85,B 0,C 180,E1 -22432.802,E2 -22432.802} C_VEL
LIN {X 0,Y 184.975,Z 671.703,A -85,B 0,C 180,E1 -22437.125,E2 -22437.125} C_VEL
LIN {X 0,Y 190.251,Z 665.585,A -85,B 0,C 180,E1 -22441.83,E2 -22441.83} C_VEL
LIN {X 0,Y 196.646,Z 658.081,A -85,B 0,C 180,E1 -22446.136,E2 -22446.136} C_VEL
LIN {X 0,Y 203.318,Z 649.936,A -85,B 0,C 180,E1 -22449.754,E2 -22449.754} C_VEL
LIN {X 0,Y 210.637,Z 640.307,A -85,B 0,C 180,E1 -22453.157,E2 -22453.157} C_VEL
LIN {X 0,Y 217.674,Z 630.426,A -85,B 0,C 180,E1 -22455.921,E2 -22455.921} C_VEL
LIN {X 0,Y 225.314,Z 618.806,A -85,B 0,C 180,E1 -22458.471,E2 -22458.471} C_VEL
LIN {X 0,Y 232.471,Z 606.652,A -85,B 0,C 180,E1 -22460.627,E2 -22460.627} C_VEL
LIN {X 0,Y 239.325,Z 593.755,A -85,B 0,C 180,E1 -22462.456,E2 -22462.456} C_VEL
LIN {X 0,Y 246.221,Z 578.986,A -85,B 0,C 180,E1 -22464.088,E2 -22464.088} C_VEL
LIN {X 0,Y 252.604,Z 562.61,A -85,B 0,C 180,E1 -22465.511,E2 -22465.511} C_VEL
LIN {X 0,Y 257.548,Z 547.282,A -85,B 0,C 180,E1 -22466.511,E2 -22466.511} C_VEL
LIN {X 0,Y 261.708,Z 531.158,A -85,B 0,C 180,E1 -22467.307,E2 -22467.307} C_VEL
LIN {X 0,Y 264.768,Z 515.399,A -85,B 0,C 180,E1 -22467.874,E2 -22467.874} C_VEL
LIN {X 0,Y 266.843,Z 498.242,A -85,B 0,C 180,E1 -22468.347,E2 -22468.347} C_VEL
LIN {X 0,Y 273.196,Z 425.099,A -85,B 0,C 180,E1 -22470.001,E2 -22470.001} C_VEL
LIN {X 0,Y 268.599,Z 414.721,A -85,B 0,C 180,E1 -22472.983,E2 -22472.983} C_VEL
LIN {X 0,Y 264.866,Z 407.182,A -85,B 0,C 180,E1 -22475.768,E2 -22475.768} C_VEL
LIN {X 0,Y 262.608,Z 403.007,A -85,B 0,C 180,E1 -22477.692,E2 -22477.692} C_VEL
LIN {X 0,Y 260.386,Z 399.473,A -85,B 0,C 180,E1 -22479.814,E2 -22479.814} C_VEL
LIN {X 0,Y 258.132,Z 395.757,A -85,B 0,C 180,E1 -22482.415,E2 -22482.415} C_VEL
LIN {X 0,Y 255.951,Z 392.19,A -85,B 0,C 180,E1 -22485.793,E2 -22485.793} C_VEL
LIN {X 0,Y 255.614,Z 391.542,A -85,B 0,C 180,E1 -22486.475,E2 -22486.475} C_VEL
LIN {X 0,Y 253.801,Z 389.091,A -85,B 0,C 180,E1 -22492.999,E2 -22492.999} C_VEL
LIN {X 0,Y 254.313,Z 389.869,A -85,B 0,C 180,E1 -22497.625,E2 -22497.625} C_VEL
LIN {X 0,Y 255.953,Z 391.779,A -85,B 0,C 180,E1 -22501.574,E2 -22501.574} C_VEL
LIN {X 0,Y 258.622,Z 396.387,A -85,B 0,C 180,E1 -22505.63,E2 -22505.63} C_VEL
LIN {X 0,Y 261.342,Z 400.851,A -85,B 0,C 180,E1 -22508.568,E2 -22508.568} C_VEL
LIN {X 0,Y 264.105,Z 405.454,A -85,B 0,C 180,E1 -22511.027,E2 -22511.027} C_VEL
LIN {X 0,Y 267.851,Z 411.919,A -85,B 0,C 180,E1 -22513.846,E2 -22513.846} C_VEL
LIN {X 0,Y 271.913,Z 419.206,A -85,B 0,C 180,E1 -22516.461,E2 -22516.461} C_VEL
LIN {X 0,Y 273.417,Z 422.083,A -85,B 0,C 180,E1 -22517.356,E2 -22517.356} C_VEL
LIN {X 0,Y 266.43,Z 500.503,A -85,B 0,C 180,E1 -22519.147,E2 -22519.147} C_VEL
LIN {X 0,Y 263.761,Z 516.83,A -85,B 0,C 180,E1 -22519.652,E2 -22519.652} C_VEL
LIN {X 0,Y 260.554,Z 531.757,A -85,B 0,C 180,E1 -22520.367,E2 -22520.367} C_VEL
LIN {X 0,Y 256.069,Z 547.712,A -85,B 0,C 180,E1 -22521.339,E2 -22521.339} C_VEL
LIN {X 0,Y 251.04,Z 562.323,A -85,B 0,C 180,E1 -22522.503,E2 -22522.503} C_VEL
LIN {X 0,Y 245.138,Z 576.694,A -85,B 0,C 180,E1 -22523.958,E2 -22523.958} C_VEL
LIN {X 0,Y 238.762,Z 590.109,A -85,B 0,C 180,E1 -22525.65,E2 -22525.65} C_VEL
LIN {X 0,Y 231.877,Z 602.796,A -85,B 0,C 180,E1 -22527.619,E2 -22527.619} C_VEL
LIN {X 0,Y 224.801,Z 614.498,A -85,B 0,C 180,E1 -22529.904,E2 -22529.904} C_VEL
LIN {X 0,Y 217.088,Z 625.878,A -85,B 0,C 180,E1 -22532.677,E2 -22532.677} C_VEL
LIN {X 0,Y 209.825,Z 635.666,A -85,B 0,C 180,E1 -22535.684,E2 -22535.684} C_VEL
LIN {X 0,Y 202.913,Z 644.352,A -85,B 0,C 180,E1 -22539.045,E2 -22539.045} C_VEL
LIN {X 0,Y 196.318,Z 652.054,A -85,B 0,C 180,E1 -22542.859,E2 -22542.859} C_VEL
LIN {X 0,Y 190.617,Z 658.432,A -85,B 0,C 180,E1 -22546.994,E2 -22546.994} C_VEL
LIN {X 0,Y 185.745,Z 663.628,A -85,B 0,C 180,E1 -22551.368,E2 -22551.368} C_VEL
LIN {X 0,Y 182.743,Z 666.701,A -85,B 0,C 180,E1 -22554.768,E2 -22554.768} C_VEL
LIN {X 0,Y 179.673,Z 669.861,A -85,B 0,C 180,E1 -22559.436,E2 -22559.436} C_VEL
LIN {X 0,Y 177.529,Z 671.848,A -85,B 0,C 180,E1 -22564.185,E2 -22564.185} C_VEL
LIN {X 0,Y 176.256,Z 672.853,A -85,B 0,C 180,E1 -22568.969,E2 -22568.969} C_VEL
LIN {X 0,Y 175.789,Z 672.812,A -85,B 0,C 180,E1 -22573.748,E2 -22573.748} C_VEL
LIN {X 0,Y 175.607,Z 671.804,A -85,B 0,C 180,E1 -22578.457,E2 -22578.457} C_VEL
LIN {X 0,Y 175.972,Z 669.818,A -85,B 0,C 180,E1 -22583.118,E2 -22583.118} C_VEL
LIN {X 0,Y 176.403,Z 668.429,A -85,B 0,C 180,E1 -22585.429,E2 -22585.429} C_VEL
LIN {X 0,Y 177.258,Z 664.982,A -85,B 0,C 180,E1 -22590,E2 -22590} C_VEL
LIN {X 0,Y 178.873,Z 660.422,A -85,B 0,C 180,E1 -22594.507,E2 -22594.507} C_VEL
LIN {X 0,Y 181.184,Z 654.769,A -85,B 0,C 180,E1 -22598.926,E2 -22598.926} C_VEL
LIN {X 0,Y 184.487,Z 647.911,A -85,B 0,C 180,E1 -22603.213,E2 -22603.213} C_VEL
LIN {X 0,Y 188.61,Z 639.584,A -85,B 0,C 180,E1 -22607.343,E2 -22607.343} C_VEL
LIN {X 0,Y 193.612,Z 629.688,A -85,B 0,C 180,E1 -22611.284,E2 -22611.284} C_VEL
LIN {X 0,Y 198.519,Z 619.532,A -85,B 0,C 180,E1 -22614.58,E2 -22614.58} C_VEL
LIN {X 0,Y 203.913,Z 607.648,A -85,B 0,C 180,E1 -22617.729,E2 -22617.729} C_VEL
LIN {X 0,Y 209.358,Z 594.569,A -85,B 0,C 180,E1 -22620.513,E2 -22620.513} C_VEL
LIN {X 0,Y 214.313,Z 581.477,A -85,B 0,C 180,E1 -22622.757,E2 -22622.757} C_VEL
LIN {X 0,Y 219.114,Z 567.403,A -85,B 0,C 180,E1 -22624.703,E2 -22624.703} C_VEL
LIN {X 0,Y 222.97,Z 554.105,A -85,B 0,C 180,E1 -22626.228,E2 -22626.228} C_VEL
LIN {X 0,Y 226.518,Z 539.796,A -85,B 0,C 180,E1 -22627.509,E2 -22627.509} C_VEL
LIN {X 0,Y 229.946,Z 522.965,A -85,B 0,C 180,E1 -22628.656,E2 -22628.656} C_VEL
LIN {X 0,Y 232.541,Z 506.048,A -85,B 0,C 180,E1 -22629.466,E2 -22629.466} C_VEL
LIN {X 0,Y 234.261,Z 488.385,A -85,B 0,C 180,E1 -22630.026,E2 -22630.026} C_VEL
LIN {X 0,Y 240.543,Z 399.417,A -85,B 0,C 180,E1 -22632.345,E2 -22632.345} C_VEL
LIN {X 0,Y 239.033,Z 395.942,A -85,B 0,C 180,E1 -22632.944,E2 -22632.944} C_VEL
LIN {X 0,Y 232.164,Z 382.922,A -85,B 0,C 180,E1 -22635.728,E2 -22635.728} C_VEL
LIN {X 0,Y 226.405,Z 373.2,A -85,B 0,C 180,E1 -22638.273,E2 -22638.273} C_VEL
LIN {X 0,Y 219.863,Z 362.972,A -85,B 0,C 180,E1 -22641.506,E2 -22641.506} C_VEL
LIN {X 0,Y 213.633,Z 354.104,A -85,B 0,C 180,E1 -22645.035,E2 -22645.035} C_VEL
LIN {X 0,Y 210.901,Z 350.279,A -85,B 0,C 180,E1 -22646.785,E2 -22646.785} C_VEL
LIN {X 0,Y 207.579,Z 345.938,A -85,B 0,C 180,E1 -22649.118,E2 -22649.118} C_VEL
LIN {X 0,Y 204.649,Z 342.122,A -85,B 0,C 180,E1 -22651.425,E2 -22651.425} C_VEL
LIN {X 0,Y 203.664,Z 341.025,A -85,B 0,C 180,E1 -22652.253,E2 -22652.253} C_VEL
LIN {X 0,Y 201.15,Z 338.139,A -85,B 0,C 180,E1 -22654.578,E2 -22654.578} C_VEL
LIN {X 0,Y 200.111,Z 336.269,A -85,B 0,C 180,E1 -22655.727,E2 -22655.727} C_VEL
LIN {X 0,Y 197.183,Z 333.668,A -85,B 0,C 180,E1 -22659.118,E2 -22659.118} C_VEL
LIN {X 0,Y 195.655,Z 330.697,A -85,B 0,C 180,E1 -22661.594,E2 -22661.594} C_VEL
LIN {X 0,Y 192.16,Z 327.502,A -85,B 0,C 180,E1 -22671.587,E2 -22671.587} C_VEL
LIN {X 0,Y 192.4,Z 327.768,A -85,B 0,C 180,E1 -22676.858,E2 -22676.858} C_VEL
LIN {X 0,Y 193.332,Z 328.706,A -85,B 0,C 180,E1 -22680.324,E2 -22680.324} C_VEL
LIN {X 0,Y 195.75,Z 330.612,A -85,B 0,C 180,E1 -22685.149,E2 -22685.149} C_VEL
LIN {X 0,Y 196.245,Z 331.033,A -85,B 0,C 180,E1 -22685.909,E2 -22685.909} C_VEL
LIN {X 0,Y 197.734,Z 333.912,A -85,B 0,C 180,E1 -22688.172,E2 -22688.172} C_VEL
LIN {X 0,Y 200.004,Z 336.058,A -85,B 0,C 180,E1 -22690.758,E2 -22690.758} C_VEL
LIN {X 0,Y 200.575,Z 336.756,A -85,B 0,C 180,E1 -22691.366,E2 -22691.366} C_VEL
LIN {X 0,Y 202.925,Z 340.21,A -85,B 0,C 180,E1 -22693.71,E2 -22693.71} C_VEL
LIN {X 0,Y 204.511,Z 341.747,A -85,B 0,C 180,E1 -22695.054,E2 -22695.054} C_VEL
LIN {X 0,Y 207.359,Z 345.703,A -85,B 0,C 180,E1 -22697.341,E2 -22697.341} C_VEL
LIN {X 0,Y 208.63,Z 347.23,A -85,B 0,C 180,E1 -22698.258,E2 -22698.258} C_VEL
LIN {X 0,Y 212.284,Z 352.148,A -85,B 0,C 180,E1 -22700.721,E2 -22700.721} C_VEL
LIN {X 0,Y 215.899,Z 357.23,A -85,B 0,C 180,E1 -22702.923,E2 -22702.923} C_VEL
LIN {X 0,Y 220.491,Z 363.923,A -85,B 0,C 180,E1 -22705.439,E2 -22705.439} C_VEL
LIN {X 0,Y 226.895,Z 373.803,A -85,B 0,C 180,E1 -22708.553,E2 -22708.553} C_VEL
LIN {X 0,Y 231.754,Z 383.447,A -85,B 0,C 180,E1 -22710.779,E2 -22710.779} C_VEL
LIN {X 0,Y 235.531,Z 391.563,A -85,B 0,C 180,E1 -22712.404,E2 -22712.404} C_VEL
LIN {X 0,Y 236.487,Z 394.84,A -85,B 0,C 180,E1 -22712.857,E2 -22712.857} C_VEL
LIN {X 0,Y 236.91,Z 398.521,A -85,B 0,C 180,E1 -22713.161,E2 -22713.161} C_VEL
LIN {X 0,Y 236.798,Z 404.404,A -85,B 0,C 180,E1 -22713.409,E2 -22713.409} C_VEL
LIN {X 0,Y 234.472,Z 423.071,A -85,B 0,C 180,E1 -22713.607,E2 -22713.607} C_VEL
LIN {X 0,Y 228.186,Z 508.029,A -85,B 0,C 180,E1 -22715.881,E2 -22715.881} C_VEL
LIN {X 0,Y 225.875,Z 524.958,A -85,B 0,C 180,E1 -22716.569,E2 -22716.569} C_VEL
LIN {X 0,Y 222.615,Z 541.522,A -85,B 0,C 180,E1 -22717.514,E2 -22717.514} C_VEL
LIN {X 0,Y 218.898,Z 556.643,A -85,B 0,C 180,E1 -22718.686,E2 -22718.686} C_VEL
LIN {X 0,Y 214.817,Z 570.854,A -85,B 0,C 180,E1 -22720.116,E2 -22720.116} C_VEL
LIN {X 0,Y 209.92,Z 584.826,A -85,B 0,C 180,E1 -22721.848,E2 -22721.848} C_VEL
LIN {X 0,Y 204.419,Z 599.233,A -85,B 0,C 180,E1 -22724.136,E2 -22724.136} C_VEL
LIN {X 0,Y 198.697,Z 612.457,A -85,B 0,C 180,E1 -22726.741,E2 -22726.741} C_VEL
LIN {X 0,Y 193.4,Z 623.947,A -85,B 0,C 180,E1 -22729.544,E2 -22729.544} C_VEL
LIN {X 0,Y 187.599,Z 635.816,A -85,B 0,C 180,E1 -22733.173,E2 -22733.173} C_VEL
LIN {X 0,Y 182.088,Z 646.547,A -85,B 0,C 180,E1 -22737.293,E2 -22737.293} C_VEL
LIN {X 0,Y 177.617,Z 655.527,A -85,B 0,C 180,E1 -22741.653,E2 -22741.653} C_VEL
LIN {X 0,Y 174.081,Z 663.012,A -85,B 0,C 180,E1 -22746.189,E2 -22746.189} C_VEL
LIN {X 0,Y 171.518,Z 669.177,A -85,B 0,C 180,E1 -22750.865,E2 -22750.865} C_VEL
LIN {X 0,Y 169.883,Z 674.047,A -85,B 0,C 180,E1 -22755.628,E2 -22755.628} C_VEL
LIN {X 0,Y 169.025,Z 677.855,A -85,B 0,C 180,E1 -22760.426,E2 -22760.426} C_VEL
LIN {X 0,Y 168.924,Z 680.528,A -85,B 0,C 180,E1 -22765.227,E2 -22765.227} C_VEL
LIN {X 0,Y 169.011,Z 682.21,A -85,B 0,C 180,E1 -22770,E2 -22770} C_VEL
LIN {X 0,Y 168.842,Z 682.835,A -85,B 0,C 180,E1 -22774.776,E2 -22774.776} C_VEL
LIN {X 0,Y 169.034,Z 682.548,A -85,B 0,C 180,E1 -22779.574,E2 -22779.574} C_VEL
LIN {X 0,Y 169.964,Z 681.26,A -85,B 0,C 180,E1 -22784.365,E2 -22784.365} C_VEL
LIN {X 0,Y 171.881,Z 679.094,A -85,B 0,C 180,E1 -22789.094,E2 -22789.094} C_VEL
LIN {X 0,Y 174.729,Z 675.881,A -85,B 0,C 180,E1 -22793.718,E2 -22793.718} C_VEL
LIN {X 0,Y 179.75,Z 670.481,A -85,B 0,C 180,E1 -22799.258,E2 -22799.258} C_VEL
LIN {X 0,Y 184.68,Z 665.141,A -85,B 0,C 180,E1 -22803.36,E2 -22803.36} C_VEL
LIN {X 0,Y 190.922,Z 658.217,A -85,B 0,C 180,E1 -22807.401,E2 -22807.401} C_VEL
LIN {X 0,Y 197.87,Z 650.154,A -85,B 0,C 180,E1 -22811.079,E2 -22811.079} C_VEL
LIN {X 0,Y 205.487,Z 640.615,A -85,B 0,C 180,E1 -22814.518,E2 -22814.518} C_VEL
LIN {X 0,Y 213.895,Z 629.29,A -85,B 0,C 180,E1 -22817.671,E2 -22817.671} C_VEL
LIN {X 0,Y 221.89,Z 617.529,A -85,B 0,C 180,E1 -22820.182,E2 -22820.182} C_VEL
LIN {X 0,Y 228.796,Z 606.023,A -85,B 0,C 180,E1 -22822.191,E2 -22822.191} C_VEL
LIN {X 0,Y 235.763,Z 593.289,A -85,B 0,C 180,E1 -22823.959,E2 -22823.959} C_VEL
LIN {X 0,Y 242.166,Z 579.909,A -85,B 0,C 180,E1 -22825.435,E2 -22825.435} C_VEL
LIN {X 0,Y 248.021,Z 565.538,A -85,B 0,C 180,E1 -22826.712,E2 -22826.712} C_VEL
LIN {X 0,Y 253.415,Z 549.957,A -85,B 0,C 180,E1 -22827.765,E2 -22827.765} C_VEL
LIN {X 0,Y 257.827,Z 534.089,A -85,B 0,C 180,E1 -22828.583,E2 -22828.583} C_VEL
LIN {X 0,Y 261.025,Z 519.131,A -85,B 0,C 180,E1 -22829.135,E2 -22829.135} C_VEL
LIN {X 0,Y 263.382,Z 502.235,A -85,B 0,C 180,E1 -22829.626,E2 -22829.626} C_VEL
LIN {X 0,Y 269.978,Z 428.664,A -85,B 0,C 180,E1 -22831.304,E2 -22831.304} C_VEL
LIN {X 0,Y 265.691,Z 418.882,A -85,B 0,C 180,E1 -22834.307,E2 -22834.307} C_VEL
LIN {X 0,Y 261.886,Z 410.889,A -85,B 0,C 180,E1 -22837.474,E2 -22837.474} C_VEL
LIN {X 0,Y 258.954,Z 406.044,A -85,B 0,C 180,E1 -22840.333,E2 -22840.333} C_VEL
LIN {X 0,Y 256.912,Z 402.551,A -85,B 0,C 180,E1 -22842.812,E2 -22842.812} C_VEL
LIN {X 0,Y 254.877,Z 399.031,A -85,B 0,C 180,E1 -22846.134,E2 -22846.134} C_VEL
LIN {X 0,Y 254.343,Z 398.332,A -85,B 0,C 180,E1 -22847.23,E2 -22847.23} C_VEL
LIN {X 0,Y 252.929,Z 396.128,A -85,B 0,C 180,E1 -22852.975,E2 -22852.975} C_VEL
LIN {X 0,Y 253.43,Z 396.934,A -85,B 0,C 180,E1 -22857.617,E2 -22857.617} C_VEL
LIN {X 0,Y 254.925,Z 398.759,A -85,B 0,C 180,E1 -22861.334,E2 -22861.334} C_VEL
LIN {X 0,Y 257.315,Z 403.016,A -85,B 0,C 180,E1 -22865.143,E2 -22865.143} C_VEL
LIN {X 0,Y 260.034,Z 407.69,A -85,B 0,C 180,E1 -22868.22,E2 -22868.22} C_VEL
LIN {X 0,Y 262.492,Z 411.908,A -85,B 0,C 180,E1 -22870.498,E2 -22870.498} C_VEL
LIN {X 0,Y 266.259,Z 418.66,A -85,B 0,C 180,E1 -22873.452,E2 -22873.452} C_VEL
LIN {X 0,Y 270.165,Z 425.969,A -85,B 0,C 180,E1 -22876.053,E2 -22876.053} C_VEL
LIN {X 0,Y 263.37,Z 500.559,A -85,B 0,C 180,E1 -22877.764,E2 -22877.764} C_VEL
LIN {X 0,Y 260.642,Z 516.943,A -85,B 0,C 180,E1 -22878.259,E2 -22878.259} C_VEL
LIN {X 0,Y 257.23,Z 532.372,A -85,B 0,C 180,E1 -22878.988,E2 -22878.988} C_VEL
LIN {X 0,Y 252.76,Z 547.869,A -85,B 0,C 180,E1 -22879.921,E2 -22879.921} C_VEL
LIN {X 0,Y 247.598,Z 562.484,A -85,B 0,C 180,E1 -22881.069,E2 -22881.069} C_VEL
LIN {X 0,Y 241.536,Z 576.862,A -85,B 0,C 180,E1 -22882.506,E2 -22882.506} C_VEL
LIN {X 0,Y 234.968,Z 590.281,A -85,B 0,C 180,E1 -22884.178,E2 -22884.178} C_VEL
LIN {X 0,Y 228.296,Z 602.293,A -85,B 0,C 180,E1 -22886.015,E2 -22886.015} C_VEL
LIN {X 0,Y 220.719,Z 614.349,A -85,B 0,C 180,E1 -22888.329,E2 -22888.329} C_VEL
LIN {X 0,Y 213.092,Z 625.263,A -85,B 0,C 180,E1 -22890.962,E2 -22890.962} C_VEL
LIN {X 0,Y 205.512,Z 635.191,A -85,B 0,C 180,E1 -22893.973,E2 -22893.973} C_VEL
LIN {X 0,Y 197.844,Z 644.399,A -85,B 0,C 180,E1 -22897.518,E2 -22897.518} C_VEL
LIN {X 0,Y 190.549,Z 652.513,A -85,B 0,C 180,E1 -22901.599,E2 -22901.599} C_VEL
LIN {X 0,Y 185.108,Z 658.247,A -85,B 0,C 180,E1 -22905.38,E2 -22905.38} C_VEL
LIN {X 0,Y 179.866,Z 663.544,A -85,B 0,C 180,E1 -22909.855,E2 -22909.855} C_VEL
LIN {X 0,Y 176.618,Z 666.665,A -85,B 0,C 180,E1 -22913.353,E2 -22913.353} C_VEL
LIN {X 0,Y 172.956,Z 670.111,A -85,B 0,C 180,E1 -22918.578,E2 -22918.578} C_VEL
LIN {X 0,Y 170.794,Z 671.952,A -85,B 0,C 180,E1 -22923.087,E2 -22923.087} C_VEL
LIN {X 0,Y 169.353,Z 673.047,A -85,B 0,C 180,E1 -22928.069,E2 -22928.069} C_VEL
LIN {X 0,Y 168.685,Z 673.022,A -85,B 0,C 180,E1 -22933.392,E2 -22933.392} C_VEL
LIN {X 0,Y 168.495,Z 672.126,A -85,B 0,C 180,E1 -22937.962,E2 -22937.962} C_VEL
LIN {X 0,Y 168.842,Z 670.18,A -85,B 0,C 180,E1 -22942.826,E2 -22942.826} C_VEL
LIN {X 0,Y 169.301,Z 668.833,A -85,B 0,C 180,E1 -22945.237,E2 -22945.237} C_VEL
LIN {X 0,Y 170.14,Z 665.473,A -85,B 0,C 180,E1 -22950,E2 -22950} C_VEL
LIN {X 0,Y 171.792,Z 660.964,A -85,B 0,C 180,E1 -22954.693,E2 -22954.693} C_VEL
LIN {X 0,Y 174.185,Z 655.41,A -85,B 0,C 180,E1 -22959.287,E2 -22959.287} C_VEL
LIN {X 0,Y 177.608,Z 648.605,A -85,B 0,C 180,E1 -22963.734,E2 -22963.734} C_VEL
LIN {X 0,Y 181.887,Z 640.389,A -85,B 0,C 180,E1 -22968.006,E2 -22968.006} C_VEL
LIN {X 0,Y 187.071,Z 630.617,A -85,B 0,C 180,E1 -22972.066,E2 -22972.066} C_VEL
LIN {X 0,Y 192.132,Z 620.609,A -85,B 0,C 180,E1 -22975.455,E2 -22975.455} C_VEL
LIN {X 0,Y 197.731,Z 608.826,A -85,B 0,C 180,E1 -22978.674,E2 -22978.674} C_VEL
LIN {X 0,Y 202.93,Z 596.96,A -85,B 0,C 180,E1 -22981.298,E2 -22981.298} C_VEL
LIN {X 0,Y 207.967,Z 584.327,A -85,B 0,C 180,E1 -22983.599,E2 -22983.599} C_VEL
LIN {X 0,Y 212.893,Z 570.812,A -85,B 0,C 180,E1 -22985.579,E2 -22985.579} C_VEL
LIN {X 0,Y 217.331,Z 556.175,A -85,B 0,C 180,E1 -22987.325,E2 -22987.325} C_VEL
LIN {X 0,Y 221.259,Z 541.252,A -85,B 0,C 180,E1 -22988.707,E2 -22988.707} C_VEL
LIN {X 0,Y 224.791,Z 524.843,A -85,B 0,C 180,E1 -22989.861,E2 -22989.861} C_VEL
LIN {X 0,Y 227.45,Z 508.754,A -85,B 0,C 180,E1 -22990.676,E2 -22990.676} C_VEL
LIN {X 0,Y 229.259,Z 492.264,A -85,B 0,C 180,E1 -22991.23,E2 -22991.23} C_VEL
LIN {X 0,Y 235.852,Z 401.834,A -85,B 0,C 180,E1 -22993.612,E2 -22993.612} C_VEL
LIN {X 0,Y 229.226,Z 388.89,A -85,B 0,C 180,E1 -22996.409,E2 -22996.409} C_VEL
LIN {X 0,Y 223.61,Z 379.04,A -85,B 0,C 180,E1 -22999.005,E2 -22999.005} C_VEL
LIN {X 0,Y 217.196,Z 368.813,A -85,B 0,C 180,E1 -23002.315,E2 -23002.315} C_VEL
LIN {X 0,Y 211.365,Z 360.265,A -85,B 0,C 180,E1 -23005.773,E2 -23005.773} C_VEL
LIN {X 0,Y 208.605,Z 356.324,A -85,B 0,C 180,E1 -23007.627,E2 -23007.627} C_VEL
LIN {X 0,Y 205.798,Z 352.496,A -85,B 0,C 180,E1 -23009.691,E2 -23009.691} C_VEL
LIN {X 0,Y 202.757,Z 348.39,A -85,B 0,C 180,E1 -23012.2,E2 -23012.2} C_VEL
LIN {X 0,Y 199.671,Z 344.85,A -85,B 0,C 180,E1 -23015.108,E2 -23015.108} C_VEL
LIN {X 0,Y 198.564,Z 342.979,A -85,B 0,C 180,E1 -23016.37,E2 -23016.37} C_VEL
LIN {X 0,Y 195.823,Z 340.302,A -85,B 0,C 180,E1 -23019.739,E2 -23019.739} C_VEL
LIN {X 0,Y 194.535,Z 337.667,A -85,B 0,C 180,E1 -23021.942,E2 -23021.942} C_VEL
LIN {X 0,Y 191.285,Z 334.568,A -85,B 0,C 180,E1 -23031.548,E2 -23031.548} C_VEL
LIN {X 0,Y 191.519,Z 334.814,A -85,B 0,C 180,E1 -23036.843,E2 -23036.843} C_VEL
LIN {X 0,Y 192.443,Z 335.808,A -85,B 0,C 180,E1 -23040.326,E2 -23040.326} C_VEL
LIN {X 0,Y 194.546,Z 337.509,A -85,B 0,C 180,E1 -23044.661,E2 -23044.661} C_VEL
LIN {X 0,Y 195.015,Z 337.961,A -85,B 0,C 180,E1 -23045.427,E2 -23045.427} C_VEL
LIN {X 0,Y 196.694,Z 341.038,A -85,B 0,C 180,E1 -23048.03,E2 -23048.03} C_VEL
LIN {X 0,Y 199.038,Z 343.387,A -85,B 0,C 180,E1 -23050.746,E2 -23050.746} C_VEL
LIN {X 0,Y 201.533,Z 347.051,A -85,B 0,C 180,E1 -23053.325,E2 -23053.325} C_VEL
LIN {X 0,Y 202.927,Z 348.569,A -85,B 0,C 180,E1 -23054.557,E2 -23054.557} C_VEL
LIN {X 0,Y 205.803,Z 352.476,A -85,B 0,C 180,E1 -23056.928,E2 -23056.928} C_VEL
LIN {X 0,Y 207.049,Z 354.25,A -85,B 0,C 180,E1 -23057.875,E2 -23057.875} C_VEL
LIN {X 0,Y 210.31,Z 358.641,A -85,B 0,C 180,E1 -23060.133,E2 -23060.133} C_VEL
LIN {X 0,Y 213.546,Z 363.344,A -85,B 0,C 180,E1 -23062.191,E2 -23062.191} C_VEL
LIN {X 0,Y 218.26,Z 370.473,A -85,B 0,C 180,E1 -23064.884,E2 -23064.884} C_VEL
LIN {X 0,Y 224.003,Z 379.64,A -85,B 0,C 180,E1 -23067.795,E2 -23067.795} C_VEL
LIN {X 0,Y 228.666,Z 389.2,A -85,B 0,C 180,E1 -23070.025,E2 -23070.025} C_VEL
LIN {X 0,Y 233.986,Z 401.439,A -85,B 0,C 180,E1 -23072.408,E2 -23072.408} C_VEL
LIN {X 0,Y 235.76,Z 405.922,A -85,B 0,C 180,E1 -23073.171,E2 -23073.171} C_VEL
LIN {X 0,Y 234.472,Z 423.071,A -85,B 0,C 180,E1 -23073.607,E2 -23073.607} C_VEL
LIN {X 0,Y 233.618,Z 428.917,A -85,B 0,C 180,E1 -23073.632,E2 -23073.632} C_VEL
LIN {X 0,Y 228.605,Z 447.953,A -85,B 0,C 180,E1 -23073.029,E2 -23073.029} C_VEL
LIN {X 0,Y 227.754,Z 453.798,A -85,B 0,C 180,E1 -23073.053,E2 -23073.053} C_VEL
LIN {X 0,Y 223.425,Z 509.138,A -85,B 0,C 180,E1 -23074.555,E2 -23074.555} C_VEL
LIN {X 0,Y 220.907,Z 526.556,A -85,B 0,C 180,E1 -23075.291,E2 -23075.291} C_VEL
LIN {X 0,Y 217.403,Z 543.255,A -85,B 0,C 180,E1 -23076.278,E2 -23076.278} C_VEL
LIN {X 0,Y 213.601,Z 557.926,A -85,B 0,C 180,E1 -23077.461,E2 -23077.461} C_VEL
LIN {X 0,Y 209.108,Z 572.684,A -85,B 0,C 180,E1 -23078.994,E2 -23078.994} C_VEL
LIN {X 0,Y 203.685,Z 587.542,A -85,B 0,C 180,E1 -23080.914,E2 -23080.914} C_VEL
LIN {X 0,Y 197.943,Z 601.708,A -85,B 0,C 180,E1 -23083.293,E2 -23083.293} C_VEL
LIN {X 0,Y 192.095,Z 614.488,A -85,B 0,C 180,E1 -23085.962,E2 -23085.962} C_VEL
LIN {X 0,Y 185.952,Z 626.958,A -85,B 0,C 180,E1 -23089.226,E2 -23089.226} C_VEL
LIN {X 0,Y 180.319,Z 637.925,A -85,B 0,C 180,E1 -23092.835,E2 -23092.835} C_VEL
LIN {X 0,Y 175.384,Z 647.133,A -85,B 0,C 180,E1 -23096.565,E2 -23096.565} C_VEL
LIN {X 0,Y 170.762,Z 655.97,A -85,B 0,C 180,E1 -23101.08,E2 -23101.08} C_VEL
LIN {X 0,Y 167.481,Z 662.497,A -85,B 0,C 180,E1 -23105.189,E2 -23105.189} C_VEL
LIN {X 0,Y 164.703,Z 668.698,A -85,B 0,C 180,E1 -23110.04,E2 -23110.04} C_VEL
LIN {X 0,Y 162.942,Z 673.638,A -85,B 0,C 180,E1 -23115.002,E2 -23115.002} C_VEL
LIN {X 0,Y 161.957,Z 677.509,A -85,B 0,C 180,E1 -23120.004,E2 -23120.004} C_VEL
LIN {X 0,Y 161.833,Z 680.216,A -85,B 0,C 180,E1 -23125.018,E2 -23125.018} C_VEL
LIN {X 0,Y 161.921,Z 681.958,A -85,B 0,C 180,E1 -23130,E2 -23130} C_VEL
LIN {X 0,Y 161.735,Z 682.611,A -85,B 0,C 180,E1 -23134.986,E2 -23134.986} C_VEL
LIN {X 0,Y 162,Z 682.383,A -85,B 0,C 180,E1 -23139.993,E2 -23139.993} C_VEL
LIN {X 0,Y 163.037,Z 681.124,A -85,B 0,C 180,E1 -23144.99,E2 -23144.99} C_VEL
LIN {X 0,Y 165.739,Z 678.288,A -85,B 0,C 180,E1 -23151.114,E2 -23151.114} C_VEL
LIN {X 0,Y 170.122,Z 673.916,A -85,B 0,C 180,E1 -23157.028,E2 -23157.028} C_VEL
LIN {X 0,Y 174.741,Z 669.262,A -85,B 0,C 180,E1 -23161.524,E2 -23161.524} C_VEL
LIN {X 0,Y 180.39,Z 663.472,A -85,B 0,C 180,E1 -23165.761,E2 -23165.761} C_VEL
LIN {X 0,Y 187.877,Z 655.536,A -85,B 0,C 180,E1 -23170.187,E2 -23170.187} C_VEL
LIN {X 0,Y 195.698,Z 646.695,A -85,B 0,C 180,E1 -23173.958,E2 -23173.958} C_VEL
LIN {X 0,Y 203.69,Z 636.916,A -85,B 0,C 180,E1 -23177.156,E2 -23177.156} C_VEL
LIN {X 0,Y 211.533,Z 626.504,A -85,B 0,C 180,E1 -23179.832,E2 -23179.832} C_VEL
LIN {X 0,Y 219.781,Z 614.355,A -85,B 0,C 180,E1 -23182.321,E2 -23182.321} C_VEL
LIN {X 0,Y 226.564,Z 603.246,A -85,B 0,C 180,E1 -23184.135,E2 -23184.135} C_VEL
LIN {X 0,Y 233.023,Z 591.546,A -85,B 0,C 180,E1 -23185.653,E2 -23185.653} C_VEL
LIN {X 0,Y 238.913,Z 579.422,A -85,B 0,C 180,E1 -23186.969,E2 -23186.969} C_VEL
LIN {X 0,Y 244.926,Z 564.982,A -85,B 0,C 180,E1 -23188.22,E2 -23188.22} C_VEL
LIN {X 0,Y 250.452,Z 549.302,A -85,B 0,C 180,E1 -23189.247,E2 -23189.247} C_VEL
LIN {X 0,Y 254.907,Z 533.397,A -85,B 0,C 180,E1 -23190.055,E2 -23190.055} C_VEL
LIN {X 0,Y 258.472,Z 516.817,A -85,B 0,C 180,E1 -23190.636,E2 -23190.636} C_VEL
LIN {X 0,Y 260.742,Z 499.686,A -85,B 0,C 180,E1 -23191.11,E2 -23191.11} C_VEL
LIN {X 0,Y 266.925,Z 432.496,A -85,B 0,C 180,E1 -23192.607,E2 -23192.607} C_VEL
LIN {X 0,Y 263.429,Z 424.128,A -85,B 0,C 180,E1 -23195.266,E2 -23195.266} C_VEL
LIN {X 0,Y 259.941,Z 416.621,A -85,B 0,C 180,E1 -23198.379,E2 -23198.379} C_VEL
LIN {X 0,Y 257.518,Z 412.588,A -85,B 0,C 180,E1 -23200.884,E2 -23200.884} C_VEL
LIN {X 0,Y 255.696,Z 409.334,A -85,B 0,C 180,E1 -23203.224,E2 -23203.224} C_VEL
LIN {X 0,Y 253.616,Z 405.49,A -85,B 0,C 180,E1 -23206.911,E2 -23206.911} C_VEL
LIN {X 0,Y 252.083,Z 403.297,A -85,B 0,C 180,E1 -23212.47,E2 -23212.47} C_VEL
LIN {X 0,Y 252.051,Z 403.302,A -85,B 0,C 180,E1 -23214.665,E2 -23214.665} C_VEL
LIN {X 0,Y 252.629,Z 404.114,A -85,B 0,C 180,E1 -23217.906,E2 -23217.906} C_VEL
LIN {X 0,Y 253.848,Z 405.589,A -85,B 0,C 180,E1 -23220.968,E2 -23220.968} C_VEL
LIN {X 0,Y 256.179,Z 409.995,A -85,B 0,C 180,E1 -23224.87,E2 -23224.87} C_VEL
LIN {X 0,Y 258.623,Z 414.318,A -85,B 0,C 180,E1 -23227.749,E2 -23227.749} C_VEL
LIN {X 0,Y 260.89,Z 418.374,A -85,B 0,C 180,E1 -23229.951,E2 -23229.951} C_VEL
LIN {X 0,Y 264.23,Z 424.596,A -85,B 0,C 180,E1 -23232.713,E2 -23232.713} C_VEL
LIN {X 0,Y 267.087,Z 430.095,A -85,B 0,C 180,E1 -23234.754,E2 -23234.754} C_VEL
LIN {X 0,Y 260.463,Z 500.605,A -85,B 0,C 180,E1 -23236.347,E2 -23236.347} C_VEL
LIN {X 0,Y 257.68,Z 517.055,A -85,B 0,C 180,E1 -23236.832,E2 -23236.832} C_VEL
LIN {X 0,Y 254.197,Z 532.455,A -85,B 0,C 180,E1 -23237.545,E2 -23237.545} C_VEL
LIN {X 0,Y 249.608,Z 548.023,A -85,B 0,C 180,E1 -23238.466,E2 -23238.466} C_VEL
LIN {X 0,Y 244.315,Z 562.64,A -85,B 0,C 180,E1 -23239.593,E2 -23239.593} C_VEL
LIN {X 0,Y 237.901,Z 577.436,A -85,B 0,C 180,E1 -23241.053,E2 -23241.053} C_VEL
LIN {X 0,Y 231.335,Z 590.453,A -85,B 0,C 180,E1 -23242.66,E2 -23242.66} C_VEL
LIN {X 0,Y 224.104,Z 603.016,A -85,B 0,C 180,E1 -23244.57,E2 -23244.57} C_VEL
LIN {X 0,Y 216.797,Z 614.248,A -85,B 0,C 180,E1 -23246.708,E2 -23246.708} C_VEL
LIN {X 0,Y 209.308,Z 624.674,A -85,B 0,C 180,E1 -23249.189,E2 -23249.189} C_VEL
LIN {X 0,Y 201.292,Z 634.824,A -85,B 0,C 180,E1 -23252.215,E2 -23252.215} C_VEL
LIN {X 0,Y 193.385,Z 643.942,A -85,B 0,C 180,E1 -23255.687,E2 -23255.687} C_VEL
LIN {X 0,Y 186.38,Z 651.382,A -85,B 0,C 180,E1 -23259.376,E2 -23259.376} C_VEL
LIN {X 0,Y 179.78,Z 658.065,A -85,B 0,C 180,E1 -23263.68,E2 -23263.68} C_VEL
LIN {X 0,Y 174.119,Z 663.458,A -85,B 0,C 180,E1 -23268.241,E2 -23268.241} C_VEL
LIN {X 0,Y 170.587,Z 666.633,A -85,B 0,C 180,E1 -23271.831,E2 -23271.831} C_VEL
LIN {X 0,Y 166.807,Z 669.907,A -85,B 0,C 180,E1 -23276.789,E2 -23276.789} C_VEL
LIN {X 0,Y 164.106,Z 672.058,A -85,B 0,C 180,E1 -23281.895,E2 -23281.895} C_VEL
LIN {X 0,Y 162.463,Z 673.224,A -85,B 0,C 180,E1 -23287.087,E2 -23287.087} C_VEL
LIN {X 0,Y 161.619,Z 673.227,A -85,B 0,C 180,E1 -23293.077,E2 -23293.077} C_VEL
LIN {X 0,Y 161.396,Z 672.447,A -85,B 0,C 180,E1 -23297.424,E2 -23297.424} C_VEL
LIN {X 0,Y 161.697,Z 670.544,A -85,B 0,C 180,E1 -23302.507,E2 -23302.507} C_VEL
LIN {X 0,Y 162.203,Z 669.102,A -85,B 0,C 180,E1 -23305.261,E2 -23305.261} C_VEL
LIN {X 0,Y 163.024,Z 665.931,A -85,B 0,C 180,E1 -23310,E2 -23310} C_VEL
LIN {X 0,Y 164.717,Z 661.506,A -85,B 0,C 180,E1 -23314.895,E2 -23314.895} C_VEL
LIN {X 0,Y 167.195,Z 656.05,A -85,B 0,C 180,E1 -23319.679,E2 -23319.679} C_VEL
LIN {X 0,Y 170.748,Z 649.296,A -85,B 0,C 180,E1 -23324.297,E2 -23324.297} C_VEL
LIN {X 0,Y 175.174,Z 641.193,A -85,B 0,C 180,E1 -23328.721,E2 -23328.721} C_VEL
LIN {X 0,Y 180.536,Z 631.545,A -85,B 0,C 180,E1 -23332.91,E2 -23332.91} C_VEL
LIN {X 0,Y 185.794,Z 621.646,A -85,B 0,C 180,E1 -23336.389,E2 -23336.389} C_VEL
LIN {X 0,Y 191.606,Z 609.963,A -85,B 0,C 180,E1 -23339.681,E2 -23339.681} C_VEL
LIN {X 0,Y 196.944,Z 598.285,A -85,B 0,C 180,E1 -23342.363,E2 -23342.363} C_VEL
LIN {X 0,Y 202.159,Z 585.88,A -85,B 0,C 180,E1 -23344.699,E2 -23344.699} C_VEL
LIN {X 0,Y 207.746,Z 571.097,A -85,B 0,C 180,E1 -23346.904,E2 -23346.904} C_VEL
LIN {X 0,Y 212.899,Z 554.723,A -85,B 0,C 180,E1 -23348.844,E2 -23348.844} C_VEL
LIN {X 0,Y 216.675,Z 540.462,A -85,B 0,C 180,E1 -23350.14,E2 -23350.14} C_VEL
LIN {X 0,Y 220.31,Z 523.713,A -85,B 0,C 180,E1 -23351.295,E2 -23351.295} C_VEL
LIN {X 0,Y 223.052,Z 506.966,A -85,B 0,C 180,E1 -23352.108,E2 -23352.108} C_VEL
LIN {X 0,Y 224.874,Z 489.596,A -85,B 0,C 180,E1 -23352.672,E2 -23352.672} C_VEL
LIN {X 0,Y 231.24,Z 404.649,A -85,B 0,C 180,E1 -23354.922,E2 -23354.922} C_VEL
LIN {X 0,Y 225.025,Z 392.436,A -85,B 0,C 180,E1 -23357.712,E2 -23357.712} C_VEL
LIN {X 0,Y 219.946,Z 383.447,A -85,B 0,C 180,E1 -23360.207,E2 -23360.207} C_VEL
LIN {X 0,Y 214.512,Z 374.529,A -85,B 0,C 180,E1 -23363.181,E2 -23363.181} C_VEL
LIN {X 0,Y 209.026,Z 366.274,A -85,B 0,C 180,E1 -23366.598,E2 -23366.598} C_VEL
LIN {X 0,Y 206.555,Z 362.621,A -85,B 0,C 180,E1 -23368.343,E2 -23368.343} C_VEL
LIN {X 0,Y 203.693,Z 358.689,A -85,B 0,C 180,E1 -23370.541,E2 -23370.541} C_VEL
LIN {X 0,Y 200.616,Z 354.462,A -85,B 0,C 180,E1 -23373.236,E2 -23373.236} C_VEL
LIN {X 0,Y 198.083,Z 351.322,A -85,B 0,C 180,E1 -23375.792,E2 -23375.792} C_VEL
LIN {X 0,Y 197.142,Z 349.75,A -85,B 0,C 180,E1 -23376.911,E2 -23376.911} C_VEL
LIN {X 0,Y 194.453,Z 346.901,A -85,B 0,C 180,E1 -23380.416,E2 -23380.416} C_VEL
LIN {X 0,Y 193.325,Z 344.567,A -85,B 0,C 180,E1 -23382.459,E2 -23382.459} C_VEL
LIN {X 0,Y 190.41,Z 341.635,A -85,B 0,C 180,E1 -23391.509,E2 -23391.509} C_VEL
LIN {X 0,Y 190.641,Z 341.836,A -85,B 0,C 180,E1 -23396.829,E2 -23396.829} C_VEL
LIN {X 0,Y 191.555,Z 342.899,A -85,B 0,C 180,E1 -23400.327,E2 -23400.327} C_VEL
LIN {X 0,Y 193.821,Z 344.88,A -85,B 0,C 180,E1 -23404.972,E2 -23404.972} C_VEL
LIN {X 0,Y 195.793,Z 348.318,A -85,B 0,C 180,E1 -23408.067,E2 -23408.067} C_VEL
LIN {X 0,Y 197.625,Z 350.201,A -85,B 0,C 180,E1 -23410.241,E2 -23410.241} C_VEL
LIN {X 0,Y 200.263,Z 354.009,A -85,B 0,C 180,E1 -23413.04,E2 -23413.04} C_VEL
LIN {X 0,Y 201.286,Z 355.263,A -85,B 0,C 180,E1 -23413.985,E2 -23413.985} C_VEL
LIN {X 0,Y 204.15,Z 359.143,A -85,B 0,C 180,E1 -23416.427,E2 -23416.427} C_VEL
LIN {X 0,Y 208.265,Z 365.035,A -85,B 0,C 180,E1 -23419.48,E2 -23419.48} C_VEL
LIN {X 0,Y 212.739,Z 371.661,A -85,B 0,C 180,E1 -23422.375,E2 -23422.375} C_VEL
LIN {X 0,Y 219.349,Z 382.306,A -85,B 0,C 180,E1 -23426.09,E2 -23426.09} C_VEL
LIN {X 0,Y 222.227,Z 387.648,A -85,B 0,C 180,E1 -23427.571,E2 -23427.571} C_VEL
LIN {X 0,Y 226.634,Z 397.306,A -85,B 0,C 180,E1 -23429.746,E2 -23429.746} C_VEL
LIN {X 0,Y 231.158,Z 408.41,A -85,B 0,C 180,E1 -23431.857,E2 -23431.857} C_VEL
LIN {X 0,Y 227.754,Z 453.798,A -85,B 0,C 180,E1 -23433.053,E2 -23433.053} C_VEL
LIN {X 0,Y 226.891,Z 459.644,A -85,B 0,C 180,E1 -23433.075,E2 -23433.075} C_VEL
LIN {X 0,Y 221.841,Z 478.658,A -85,B 0,C 180,E1 -23432.418,E2 -23432.418} C_VEL
LIN {X 0,Y 220.995,Z 484.502,A -85,B 0,C 180,E1 -23432.443,E2 -23432.443} C_VEL
LIN {X 0,Y 218.809,Z 509.822,A -85,B 0,C 180,E1 -23433.164,E2 -23433.164} C_VEL
LIN {X 0,Y 216.195,Z 527.175,A -85,B 0,C 180,E1 -23433.905,E2 -23433.905} C_VEL
LIN {X 0,Y 212.605,Z 543.668,A -85,B 0,C 180,E1 -23434.894,E2 -23434.894} C_VEL
LIN {X 0,Y 208.688,Z 558.19,A -85,B 0,C 180,E1 -23436.075,E2 -23436.075} C_VEL
LIN {X 0,Y 204.059,Z 572.853,A -85,B 0,C 180,E1 -23437.614,E2 -23437.614} C_VEL
LIN {X 0,Y 198.724,Z 587.025,A -85,B 0,C 180,E1 -23439.451,E2 -23439.451} C_VEL
LIN {X 0,Y 193.048,Z 600.58,A -85,B 0,C 180,E1 -23441.728,E2 -23441.728} C_VEL
LIN {X 0,Y 186.932,Z 613.51,A -85,B 0,C 180,E1 -23444.412,E2 -23444.412} C_VEL
LIN {X 0,Y 180.643,Z 625.901,A -85,B 0,C 180,E1 -23447.662,E2 -23447.662} C_VEL
LIN {X 0,Y 174.582,Z 637.183,A -85,B 0,C 180,E1 -23451.394,E2 -23451.394} C_VEL
LIN {X 0,Y 168.701,Z 647.667,A -85,B 0,C 180,E1 -23455.778,E2 -23455.778} C_VEL
LIN {X 0,Y 163.917,Z 656.403,A -85,B 0,C 180,E1 -23460.458,E2 -23460.458} C_VEL
LIN {X 0,Y 160.099,Z 663.631,A -85,B 0,C 180,E1 -23465.353,E2 -23465.353} C_VEL
LIN {X 0,Y 157.384,Z 669.589,A -85,B 0,C 180,E1 -23470.433,E2 -23470.433} C_VEL
LIN {X 0,Y 155.654,Z 674.318,A -85,B 0,C 180,E1 -23475.621,E2 -23475.621} C_VEL
LIN {X 0,Y 154.911,Z 677.148,A -85,B 0,C 180,E1 -23479.545,E2 -23479.545} C_VEL
LIN {X 0,Y 154.723,Z 679.903,A -85,B 0,C 180,E1 -23484.788,E2 -23484.788} C_VEL
LIN {X 0,Y 154.821,Z 681.702,A -85,B 0,C 180,E1 -23490,E2 -23490} C_VEL
LIN {X 0,Y 154.636,Z 682.388,A -85,B 0,C 180,E1 -23495.216,E2 -23495.216} C_VEL
LIN {X 0,Y 154.952,Z 682.205,A -85,B 0,C 180,E1 -23500.453,E2 -23500.453} C_VEL
LIN {X 0,Y 156.132,Z 680.991,A -85,B 0,C 180,E1 -23505.669,E2 -23505.669} C_VEL
LIN {X 0,Y 158.833,Z 678.427,A -85,B 0,C 180,E1 -23511.693,E2 -23511.693} C_VEL
LIN {X 0,Y 163.733,Z 673.911,A -85,B 0,C 180,E1 -23518.175,E2 -23518.175} C_VEL
LIN {X 0,Y 168.64,Z 669.291,A -85,B 0,C 180,E1 -23522.805,E2 -23522.805} C_VEL
LIN {X 0,Y 174.619,Z 663.576,A -85,B 0,C 180,E1 -23527.137,E2 -23527.137} C_VEL
LIN {X 0,Y 181.53,Z 656.702,A -85,B 0,C 180,E1 -23531.16,E2 -23531.16} C_VEL
LIN {X 0,Y 189.276,Z 648.401,A -85,B 0,C 180,E1 -23534.869,E2 -23534.869} C_VEL
LIN {X 0,Y 197.788,Z 638.59,A -85,B 0,C 180,E1 -23538.262,E2 -23538.262} C_VEL
LIN {X 0,Y 205.828,Z 628.555,A -85,B 0,C 180,E1 -23540.969,E2 -23540.969} C_VEL
LIN {X 0,Y 214.321,Z 616.768,A -85,B 0,C 180,E1 -23543.457,E2 -23543.457} C_VEL
LIN {X 0,Y 221.836,Z 604.944,A -85,B 0,C 180,E1 -23545.458,E2 -23545.458} C_VEL
LIN {X 0,Y 229.791,Z 591.086,A -85,B 0,C 180,E1 -23547.253,E2 -23547.253} C_VEL
LIN {X 0,Y 236.502,Z 577.465,A -85,B 0,C 180,E1 -23548.688,E2 -23548.688} C_VEL
LIN {X 0,Y 242.722,Z 562.678,A -85,B 0,C 180,E1 -23549.887,E2 -23549.887} C_VEL
LIN {X 0,Y 248.006,Z 547.54,A -85,B 0,C 180,E1 -23550.829,E2 -23550.829} C_VEL
LIN {X 0,Y 252.59,Z 531.02,A -85,B 0,C 180,E1 -23551.611,E2 -23551.611} C_VEL
LIN {X 0,Y 256.064,Z 514.269,A -85,B 0,C 180,E1 -23552.163,E2 -23552.163} C_VEL
LIN {X 0,Y 258.202,Z 497.689,A -85,B 0,C 180,E1 -23552.607,E2 -23552.607} C_VEL
LIN {X 0,Y 263.948,Z 436.977,A -85,B 0,C 180,E1 -23553.926,E2 -23553.926} C_VEL
LIN {X 0,Y 263.895,Z 436.046,A -85,B 0,C 180,E1 -23554.029,E2 -23554.029} C_VEL
LIN {X 0,Y 261.266,Z 429.61,A -85,B 0,C 180,E1 -23556.204,E2 -23556.204} C_VEL
LIN {X 0,Y 258.416,Z 423.155,A -85,B 0,C 180,E1 -23558.921,E2 -23558.921} C_VEL
LIN {X 0,Y 256.301,Z 419.419,A -85,B 0,C 180,E1 -23561.215,E2 -23561.215} C_VEL
LIN {X 0,Y 254.467,Z 416.064,A -85,B 0,C 180,E1 -23563.679,E2 -23563.679} C_VEL
LIN {X 0,Y 252.618,Z 412.463,A -85,B 0,C 180,E1 -23567.141,E2 -23567.141} C_VEL
LIN {X 0,Y 251.156,Z 410.169,A -85,B 0,C 180,E1 -23573.574,E2 -23573.574} C_VEL
LIN {X 0,Y 251.741,Z 411.165,A -85,B 0,C 180,E1 -23577.875,E2 -23577.875} C_VEL
LIN {X 0,Y 252.831,Z 412.573,A -85,B 0,C 180,E1 -23580.723,E2 -23580.723} C_VEL
LIN {X 0,Y 254.977,Z 416.775,A -85,B 0,C 180,E1 -23584.483,E2 -23584.483} C_VEL
LIN {X 0,Y 257.254,Z 421.01,A -85,B 0,C 180,E1 -23587.303,E2 -23587.303} C_VEL
LIN {X 0,Y 259.653,Z 425.469,A -85,B 0,C 180,E1 -23589.716,E2 -23589.716} C_VEL
LIN {X 0,Y 263.158,Z 432.308,A -85,B 0,C 180,E1 -23592.68,E2 -23592.68} C_VEL
LIN {X 0,Y 264.13,Z 434.253,A -85,B 0,C 180,E1 -23593.415,E2 -23593.415} C_VEL
LIN {X 0,Y 257.702,Z 500.825,A -85,B 0,C 180,E1 -23594.904,E2 -23594.904} C_VEL
LIN {X 0,Y 254.882,Z 517.169,A -85,B 0,C 180,E1 -23595.374,E2 -23595.374} C_VEL
LIN {X 0,Y 251.72,Z 531.082,A -85,B 0,C 180,E1 -23595.99,E2 -23595.99} C_VEL
LIN {X 0,Y 246.995,Z 547.147,A -85,B 0,C 180,E1 -23596.908,E2 -23596.908} C_VEL
LIN {X 0,Y 241.206,Z 562.803,A -85,B 0,C 180,E1 -23598.085,E2 -23598.085} C_VEL
LIN {X 0,Y 234.957,Z 576.86,A -85,B 0,C 180,E1 -23599.429,E2 -23599.429} C_VEL
LIN {X 0,Y 227.863,Z 590.623,A -85,B 0,C 180,E1 -23601.091,E2 -23601.091} C_VEL
LIN {X 0,Y 220.422,Z 603.193,A -85,B 0,C 180,E1 -23602.977,E2 -23602.977} C_VEL
LIN {X 0,Y 211.838,Z 615.954,A -85,B 0,C 180,E1 -23605.415,E2 -23605.415} C_VEL
LIN {X 0,Y 203.326,Z 627.173,A -85,B 0,C 180,E1 -23608.186,E2 -23608.186} C_VEL
LIN {X 0,Y 195.187,Z 636.835,A -85,B 0,C 180,E1 -23611.223,E2 -23611.223} C_VEL
LIN {X 0,Y 186.59,Z 646.134,A -85,B 0,C 180,E1 -23614.992,E2 -23614.992} C_VEL
LIN {X 0,Y 179.39,Z 653.376,A -85,B 0,C 180,E1 -23618.819,E2 -23618.819} C_VEL
LIN {X 0,Y 171.383,Z 660.83,A -85,B 0,C 180,E1 -23624.199,E2 -23624.199} C_VEL
LIN {X 0,Y 165.888,Z 665.563,A -85,B 0,C 180,E1 -23628.953,E2 -23628.953} C_VEL
LIN {X 0,Y 162.446,Z 668.42,A -85,B 0,C 180,E1 -23632.721,E2 -23632.721} C_VEL
LIN {X 0,Y 158.872,Z 671.168,A -85,B 0,C 180,E1 -23637.937,E2 -23637.937} C_VEL
LIN {X 0,Y 156.13,Z 673.07,A -85,B 0,C 180,E1 -23644.197,E2 -23644.197} C_VEL
LIN {X 0,Y 154.985,Z 673.566,A -85,B 0,C 180,E1 -23648.729,E2 -23648.729} C_VEL
LIN {X 0,Y 154.441,Z 673.255,A -85,B 0,C 180,E1 -23654.155,E2 -23654.155} C_VEL
LIN {X 0,Y 154.349,Z 671.937,A -85,B 0,C 180,E1 -23659.506,E2 -23659.506} C_VEL
LIN {X 0,Y 155.135,Z 669.343,A -85,B 0,C 180,E1 -23665.331,E2 -23665.331} C_VEL
LIN {X 0,Y 156.281,Z 665.398,A -85,B 0,C 180,E1 -23671.288,E2 -23671.288} C_VEL
LIN {X 0,Y 158.209,Z 660.807,A -85,B 0,C 180,E1 -23676.376,E2 -23676.376} C_VEL
LIN {X 0,Y 161.054,Z 655.079,A -85,B 0,C 180,E1 -23681.324,E2 -23681.324} C_VEL
LIN {X 0,Y 165.483,Z 647.162,A -85,B 0,C 180,E1 -23686.658,E2 -23686.658} C_VEL
LIN {X 0,Y 170.451,Z 638.651,A -85,B 0,C 180,E1 -23691.148,E2 -23691.148} C_VEL
LIN {X 0,Y 176.327,Z 628.434,A -85,B 0,C 180,E1 -23695.37,E2 -23695.37} C_VEL
LIN {X 0,Y 182.027,Z 617.897,A -85,B 0,C 180,E1 -23698.856,E2 -23698.856} C_VEL
LIN {X 0,Y 188.157,Z 605.577,A -85,B 0,C 180,E1 -23702.158,E2 -23702.158} C_VEL
LIN {X 0,Y 193.904,Z 593.18,A -85,B 0,C 180,E1 -23704.81,E2 -23704.81} C_VEL
LIN {X 0,Y 199.536,Z 579.766,A -85,B 0,C 180,E1 -23707.097,E2 -23707.097} C_VEL
LIN {X 0,Y 204.832,Z 565.181,A -85,B 0,C 180,E1 -23709.084,E2 -23709.084} C_VEL
LIN {X 0,Y 209.161,Z 551.177,A -85,B 0,C 180,E1 -23710.618,E2 -23710.618} C_VEL
LIN {X 0,Y 212.812,Z 537.439,A -85,B 0,C 180,E1 -23711.811,E2 -23711.811} C_VEL
LIN {X 0,Y 216.266,Z 521.08,A -85,B 0,C 180,E1 -23712.875,E2 -23712.875} C_VEL
LIN {X 0,Y 218.785,Z 505.193,A -85,B 0,C 180,E1 -23713.601,E2 -23713.601} C_VEL
LIN {X 0,Y 220.798,Z 484.997,A -85,B 0,C 180,E1 -23714.209,E2 -23714.209} C_VEL
LIN {X 0,Y 226.799,Z 408.168,A -85,B 0,C 180,E1 -23716.225,E2 -23716.225} C_VEL
LIN {X 0,Y 226.353,Z 406.741,A -85,B 0,C 180,E1 -23716.456,E2 -23716.456} C_VEL
LIN {X 0,Y 220.787,Z 395.668,A -85,B 0,C 180,E1 -23719.139,E2 -23719.139} C_VEL
LIN {X 0,Y 215.355,Z 386.091,A -85,B 0,C 180,E1 -23722.021,E2 -23722.021} C_VEL
LIN {X 0,Y 209.981,Z 377.212,A -85,B 0,C 180,E1 -23725.252,E2 -23725.252} C_VEL
LIN {X 0,Y 204.768,Z 369.168,A -85,B 0,C 180,E1 -23728.902,E2 -23728.902} C_VEL
LIN {X 0,Y 201.923,Z 365.198,A -85,B 0,C 180,E1 -23731.169,E2 -23731.169} C_VEL
LIN {X 0,Y 199.015,Z 361.101,A -85,B 0,C 180,E1 -23733.831,E2 -23733.831} C_VEL
LIN {X 0,Y 196.433,Z 357.666,A -85,B 0,C 180,E1 -23736.595,E2 -23736.595} C_VEL
LIN {X 0,Y 195.587,Z 356.413,A -85,B 0,C 180,E1 -23737.633,E2 -23737.633} C_VEL
LIN {X 0,Y 193.08,Z 353.431,A -85,B 0,C 180,E1 -23741.152,E2 -23741.152} C_VEL
LIN {X 0,Y 192.13,Z 351.484,A -85,B 0,C 180,E1 -23742.983,E2 -23742.983} C_VEL
LIN {X 0,Y 189.535,Z 348.705,A -85,B 0,C 180,E1 -23751.469,E2 -23751.469} C_VEL
LIN {X 0,Y 189.596,Z 348.792,A -85,B 0,C 180,E1 -23755.747,E2 -23755.747} C_VEL
LIN {X 0,Y 190.319,Z 349.471,A -85,B 0,C 180,E1 -23759.205,E2 -23759.205} C_VEL
LIN {X 0,Y 192.657,Z 351.794,A -85,B 0,C 180,E1 -23764.535,E2 -23764.535} C_VEL
LIN {X 0,Y 194.759,Z 355.404,A -85,B 0,C 180,E1 -23767.923,E2 -23767.923} C_VEL
LIN {X 0,Y 196.177,Z 356.938,A -85,B 0,C 180,E1 -23769.669,E2 -23769.669} C_VEL
LIN {X 0,Y 198.841,Z 360.792,A -85,B 0,C 180,E1 -23772.599,E2 -23772.599} C_VEL
LIN {X 0,Y 200.427,Z 363.129,A -85,B 0,C 180,E1 -23774.127,E2 -23774.127} C_VEL
LIN {X 0,Y 203.107,Z 366.867,A -85,B 0,C 180,E1 -23776.424,E2 -23776.424} C_VEL
LIN {X 0,Y 206.134,Z 371.243,A -85,B 0,C 180,E1 -23778.731,E2 -23778.731} C_VEL
LIN {X 0,Y 210.575,Z 378.059,A -85,B 0,C 180,E1 -23781.73,E2 -23781.73} C_VEL
LIN {X 0,Y 216.778,Z 388.417,A -85,B 0,C 180,E1 -23785.375,E2 -23785.375} C_VEL
LIN {X 0,Y 219.758,Z 394.273,A -85,B 0,C 180,E1 -23786.982,E2 -23786.982} C_VEL
LIN {X 0,Y 225.233,Z 407.186,A -85,B 0,C 180,E1 -23789.783,E2 -23789.783} C_VEL
LIN {X 0,Y 226.72,Z 411.011,A -85,B 0,C 180,E1 -23790.511,E2 -23790.511} C_VEL
LIN {X 0,Y 220.995,Z 484.502,A -85,B 0,C 180,E1 -23792.443,E2 -23792.443} C_VEL
LIN {X 0,Y 220.158,Z 490.345,A -85,B 0,C 180,E1 -23792.464,E2 -23792.464} C_VEL
LIN {X 0,Y 214.885,Z 509.312,A -85,B 0,C 180,E1 -23791.815,E2 -23791.815} C_VEL
LIN {X 0,Y 213.72,Z 515.106,A -85,B 0,C 180,E1 -23791.903,E2 -23791.903} C_VEL
LIN {X 0,Y 210.794,Z 531.642,A -85,B 0,C 180,E1 -23792.682,E2 -23792.682} C_VEL
LIN {X 0,Y 207.003,Z 547.594,A -85,B 0,C 180,E1 -23793.716,E2 -23793.716} C_VEL
LIN {X 0,Y 202.689,Z 562.45,A -85,B 0,C 180,E1 -23794.999,E2 -23794.999} C_VEL
LIN {X 0,Y 197.312,Z 577.839,A -85,B 0,C 180,E1 -23796.734,E2 -23796.734} C_VEL
LIN {X 0,Y 191.573,Z 591.952,A -85,B 0,C 180,E1 -23798.767,E2 -23798.767} C_VEL
LIN {X 0,Y 185.579,Z 605.164,A -85,B 0,C 180,E1 -23801.177,E2 -23801.177} C_VEL
LIN {X 0,Y 179.951,Z 616.53,A -85,B 0,C 180,E1 -23803.738,E2 -23803.738} C_VEL
LIN {X 0,Y 173.306,Z 628.799,A -85,B 0,C 180,E1 -23807.215,E2 -23807.215} C_VEL
LIN {X 0,Y 167.332,Z 639.217,A -85,B 0,C 180,E1 -23810.95,E2 -23810.95} C_VEL
LIN {X 0,Y 161.4,Z 649.313,A -85,B 0,C 180,E1 -23815.524,E2 -23815.524} C_VEL
LIN {X 0,Y 156.551,Z 657.77,A -85,B 0,C 180,E1 -23820.408,E2 -23820.408} C_VEL
LIN {X 0,Y 152.711,Z 664.759,A -85,B 0,C 180,E1 -23825.532,E2 -23825.532} C_VEL
LIN {X 0,Y 150.038,Z 670.411,A -85,B 0,C 180,E1 -23830.86,E2 -23830.86} C_VEL
LIN {X 0,Y 148.339,Z 674.941,A -85,B 0,C 180,E1 -23836.297,E2 -23836.297} C_VEL
LIN {X 0,Y 147.638,Z 678.298,A -85,B 0,C 180,E1 -23841.79,E2 -23841.79} C_VEL
LIN {X 0,Y 147.64,Z 680.636,A -85,B 0,C 180,E1 -23847.272,E2 -23847.272} C_VEL
LIN {X 0,Y 147.722,Z 681.427,A -85,B 0,C 180,E1 -23850,E2 -23850} C_VEL
LIN {X 0,Y 147.54,Z 682.164,A -85,B 0,C 180,E1 -23855.467,E2 -23855.467} C_VEL
LIN {X 0,Y 147.926,Z 682.012,A -85,B 0,C 180,E1 -23860.956,E2 -23860.956} C_VEL
LIN {X 0,Y 149.225,Z 680.857,A -85,B 0,C 180,E1 -23866.415,E2 -23866.415} C_VEL
LIN {X 0,Y 151.963,Z 678.552,A -85,B 0,C 180,E1 -23872.341,E2 -23872.341} C_VEL
LIN {X 0,Y 157.422,Z 673.908,A -85,B 0,C 180,E1 -23879.412,E2 -23879.412} C_VEL
LIN {X 0,Y 163.782,Z 668.368,A -85,B 0,C 180,E1 -23885.056,E2 -23885.056} C_VEL
LIN {X 0,Y 170.69,Z 662.082,A -85,B 0,C 180,E1 -23889.658,E2 -23889.658} C_VEL
LIN {X 0,Y 178.161,Z 654.922,A -85,B 0,C 180,E1 -23893.657,E2 -23893.657} C_VEL
LIN {X 0,Y 185.908,Z 646.935,A -85,B 0,C 180,E1 -23897.122,E2 -23897.122} C_VEL
LIN {X 0,Y 194.274,Z 637.58,A -85,B 0,C 180,E1 -23900.241,E2 -23900.241} C_VEL
LIN {X 0,Y 202.672,Z 627.383,A -85,B 0,C 180,E1 -23902.899,E2 -23902.899} C_VEL
LIN {X 0,Y 211.422,Z 615.488,A -85,B 0,C 180,E1 -23905.36,E2 -23905.36} C_VEL
LIN {X 0,Y 219.285,Z 603.464,A -85,B 0,C 180,E1 -23907.279,E2 -23907.279} C_VEL
LIN {X 0,Y 227.388,Z 589.359,A -85,B 0,C 180,E1 -23909.058,E2 -23909.058} C_VEL
LIN {X 0,Y 234.358,Z 575.377,A -85,B 0,C 180,E1 -23910.42,E2 -23910.42} C_VEL
LIN {X 0,Y 239.992,Z 562.123,A -85,B 0,C 180,E1 -23911.466,E2 -23911.466} C_VEL
LIN {X 0,Y 245.398,Z 546.885,A -85,B 0,C 180,E1 -23912.378,E2 -23912.378} C_VEL
LIN {X 0,Y 249.918,Z 530.855,A -85,B 0,C 180,E1 -23913.114,E2 -23913.114} C_VEL
LIN {X 0,Y 253.319,Z 514.961,A -85,B 0,C 180,E1 -23913.629,E2 -23913.629} C_VEL
LIN {X 0,Y 255.538,Z 498.625,A -85,B 0,C 180,E1 -23914.063,E2 -23914.063} C_VEL
LIN {X 0,Y 261.226,Z 440.208,A -85,B 0,C 180,E1 -23915.322,E2 -23915.322} C_VEL
LIN {X 0,Y 259.208,Z 435.141,A -85,B 0,C 180,E1 -23917.135,E2 -23917.135} C_VEL
LIN {X 0,Y 256.866,Z 429.572,A -85,B 0,C 180,E1 -23919.525,E2 -23919.525} C_VEL
LIN {X 0,Y 254.941,Z 426.021,A -85,B 0,C 180,E1 -23921.731,E2 -23921.731} C_VEL
LIN {X 0,Y 253.311,Z 422.896,A -85,B 0,C 180,E1 -23924.05,E2 -23924.05} C_VEL
LIN {X 0,Y 251.565,Z 419.405,A -85,B 0,C 180,E1 -23927.497,E2 -23927.497} C_VEL
LIN {X 0,Y 250.281,Z 417.218,A -85,B 0,C 180,E1 -23933.552,E2 -23933.552} C_VEL
LIN {X 0,Y 250.719,Z 418.026,A -85,B 0,C 180,E1 -23937.339,E2 -23937.339} C_VEL
LIN {X 0,Y 251.833,Z 419.553,A -85,B 0,C 180,E1 -23940.501,E2 -23940.501} C_VEL
LIN {X 0,Y 253.778,Z 423.579,A -85,B 0,C 180,E1 -23944.086,E2 -23944.086} C_VEL
LIN {X 0,Y 255.829,Z 427.519,A -85,B 0,C 180,E1 -23946.763,E2 -23946.763} C_VEL
LIN {X 0,Y 258.492,Z 432.614,A -85,B 0,C 180,E1 -23949.538,E2 -23949.538} C_VEL
LIN {X 0,Y 261.336,Z 438.54,A -85,B 0,C 180,E1 -23952.053,E2 -23952.053} C_VEL
LIN {X 0,Y 255.033,Z 501.645,A -85,B 0,C 180,E1 -23953.443,E2 -23953.443} C_VEL
LIN {X 0,Y 252.058,Z 518.234,A -85,B 0,C 180,E1 -23953.914,E2 -23953.914} C_VEL
LIN {X 0,Y 248.537,Z 532.989,A -85,B 0,C 180,E1 -23954.581,E2 -23954.581} C_VEL
LIN {X 0,Y 244.058,Z 547.66,A -85,B 0,C 180,E1 -23955.406,E2 -23955.406} C_VEL
LIN {X 0,Y 238.264,Z 562.963,A -85,B 0,C 180,E1 -23956.534,E2 -23956.534} C_VEL
LIN {X 0,Y 231.431,Z 577.913,A -85,B 0,C 180,E1 -23957.942,E2 -23957.942} C_VEL
LIN {X 0,Y 224.565,Z 590.792,A -85,B 0,C 180,E1 -23959.473,E2 -23959.473} C_VEL
LIN {X 0,Y 216.929,Z 603.373,A -85,B 0,C 180,E1 -23961.34,E2 -23961.34} C_VEL
LIN {X 0,Y 208.843,Z 615.022,A -85,B 0,C 180,E1 -23963.505,E2 -23963.505} C_VEL
LIN {X 0,Y 199.869,Z 626.583,A -85,B 0,C 180,E1 -23966.277,E2 -23966.277} C_VEL
LIN {X 0,Y 191.361,Z 636.382,A -85,B 0,C 180,E1 -23969.278,E2 -23969.278} C_VEL
LIN {X 0,Y 183.446,Z 644.762,A -85,B 0,C 180,E1 -23972.558,E2 -23972.558} C_VEL
LIN {X 0,Y 175.158,Z 652.696,A -85,B 0,C 180,E1 -23976.632,E2 -23976.632} C_VEL
LIN {X 0,Y 167.894,Z 659.182,A -85,B 0,C 180,E1 -23981.107,E2 -23981.107} C_VEL
LIN {X 0,Y 161.633,Z 664.399,A -85,B 0,C 180,E1 -23985.917,E2 -23985.917} C_VEL
LIN {X 0,Y 156.483,Z 668.39,A -85,B 0,C 180,E1 -23991.04,E2 -23991.04} C_VEL
LIN {X 0,Y 152.528,Z 671.229,A -85,B 0,C 180,E1 -23996.432,E2 -23996.432} C_VEL
LIN {X 0,Y 149.75,Z 673.058,A -85,B 0,C 180,E1 -24002.01,E2 -24002.01} C_VEL
LIN {X 0,Y 148.063,Z 673.76,A -85,B 0,C 180,E1 -24007.683,E2 -24007.683} C_VEL
LIN {X 0,Y 147.393,Z 673.534,A -85,B 0,C 180,E1 -24013.375,E2 -24013.375} C_VEL
LIN {X 0,Y 147.233,Z 672.255,A -85,B 0,C 180,E1 -24018.992,E2 -24018.992} C_VEL
LIN {X 0,Y 148.054,Z 669.549,A -85,B 0,C 180,E1 -24025.47,E2 -24025.47} C_VEL
LIN {X 0,Y 149.158,Z 665.888,A -85,B 0,C 180,E1 -24031.35,E2 -24031.35} C_VEL
LIN {X 0,Y 151.175,Z 661.34,A -85,B 0,C 180,E1 -24036.674,E2 -24036.674} C_VEL
LIN {X 0,Y 154.114,Z 655.71,A -85,B 0,C 180,E1 -24041.842,E2 -24041.842} C_VEL
LIN {X 0,Y 158.161,Z 648.865,A -85,B 0,C 180,E1 -24046.788,E2 -24046.788} C_VEL
LIN {X 0,Y 163.21,Z 640.559,A -85,B 0,C 180,E1 -24051.47,E2 -24051.47} C_VEL
LIN {X 0,Y 169.168,Z 630.694,A -85,B 0,C 180,E1 -24055.863,E2 -24055.863} C_VEL
LIN {X 0,Y 175.006,Z 620.567,A -85,B 0,C 180,E1 -24059.468,E2 -24059.468} C_VEL
LIN {X 0,Y 181.329,Z 608.714,A -85,B 0,C 180,E1 -24062.862,E2 -24062.862} C_VEL
LIN {X 0,Y 187.67,Z 595.658,A -85,B 0,C 180,E1 -24065.812,E2 -24065.812} C_VEL
LIN {X 0,Y 193.426,Z 582.594,A -85,B 0,C 180,E1 -24068.147,E2 -24068.147} C_VEL
LIN {X 0,Y 198.897,Z 568.573,A -85,B 0,C 180,E1 -24070.155,E2 -24070.155} C_VEL
LIN {X 0,Y 203.315,Z 555.293,A -85,B 0,C 180,E1 -24071.714,E2 -24071.714} C_VEL
LIN {X 0,Y 207.331,Z 541.067,A -85,B 0,C 180,E1 -24073.014,E2 -24073.014} C_VEL
LIN {X 0,Y 211.181,Z 524.377,A -85,B 0,C 180,E1 -24074.17,E2 -24074.17} C_VEL
LIN {X 0,Y 214.069,Z 507.755,A -85,B 0,C 180,E1 -24074.982,E2 -24074.982} C_VEL
LIN {X 0,Y 216.016,Z 490.563,A -85,B 0,C 180,E1 -24075.539,E2 -24075.539} C_VEL
LIN {X 0,Y 222.429,Z 410.655,A -85,B 0,C 180,E1 -24077.653,E2 -24077.653} C_VEL
LIN {X 0,Y 216.89,Z 399.48,A -85,B 0,C 180,E1 -24080.499,E2 -24080.499} C_VEL
LIN {X 0,Y 211.505,Z 389.754,A -85,B 0,C 180,E1 -24083.585,E2 -24083.585} C_VEL
LIN {X 0,Y 206.314,Z 381.185,A -85,B 0,C 180,E1 -24086.972,E2 -24086.972} C_VEL
LIN {X 0,Y 202.435,Z 375.026,A -85,B 0,C 180,E1 -24089.902,E2 -24089.902} C_VEL
LIN {X 0,Y 200.095,Z 371.609,A -85,B 0,C 180,E1 -24091.88,E2 -24091.88} C_VEL
LIN {X 0,Y 197.296,Z 367.589,A -85,B 0,C 180,E1 -24094.575,E2 -24094.575} C_VEL
LIN {X 0,Y 194.729,Z 363.826,A -85,B 0,C 180,E1 -24097.529,E2 -24097.529} C_VEL
LIN {X 0,Y 191.675,Z 359.811,A -85,B 0,C 180,E1 -24102.026,E2 -24102.026} C_VEL
LIN {X 0,Y 190.997,Z 358.399,A -85,B 0,C 180,E1 -24103.43,E2 -24103.43} C_VEL
LIN {X 0,Y 188.661,Z 355.765,A -85,B 0,C 180,E1 -24111.429,E2 -24111.429} C_VEL
LIN {X 0,Y 188.717,Z 355.837,A -85,B 0,C 180,E1 -24115.727,E2 -24115.727} C_VEL
LIN {X 0,Y 189.486,Z 356.666,A -85,B 0,C 180,E1 -24119.401,E2 -24119.401} C_VEL
LIN {X 0,Y 191.511,Z 358.727,A -85,B 0,C 180,E1 -24124.109,E2 -24124.109} C_VEL
LIN {X 0,Y 193.865,Z 362.63,A -85,B 0,C 180,E1 -24127.96,E2 -24127.96} C_VEL
LIN {X 0,Y 194.854,Z 363.821,A -85,B 0,C 180,E1 -24129.22,E2 -24129.22} C_VEL
LIN {X 0,Y 197.446,Z 367.591,A -85,B 0,C 180,E1 -24132.167,E2 -24132.167} C_VEL
LIN {X 0,Y 201.25,Z 373.291,A -85,B 0,C 180,E1 -24135.734,E2 -24135.734} C_VEL
LIN {X 0,Y 204.143,Z 377.658,A -85,B 0,C 180,E1 -24138.049,E2 -24138.049} C_VEL
LIN {X 0,Y 208.044,Z 383.775,A -85,B 0,C 180,E1 -24140.807,E2 -24140.807} C_VEL
LIN {X 0,Y 213.891,Z 393.866,A -85,B 0,C 180,E1 -24144.439,E2 -24144.439} C_VEL
LIN {X 0,Y 216.245,Z 398.621,A -85,B 0,C 180,E1 -24145.787,E2 -24145.787} C_VEL
LIN {X 0,Y 221.252,Z 410.665,A -85,B 0,C 180,E1 -24148.52,E2 -24148.52} C_VEL
LIN {X 0,Y 222.375,Z 413.627,A -85,B 0,C 180,E1 -24149.106,E2 -24149.106} C_VEL
LIN {X 0,Y 214.625,Z 508.206,A -85,B 0,C 180,E1 -24151.638,E2 -24151.638} C_VEL
LIN {X 0,Y 213.72,Z 515.106,A -85,B 0,C 180,E1 -24151.903,E2 -24151.903} C_VEL
LIN {X 0,Y 212.726,Z 518.972,A -85,B 0,C 180,E1 -24151.907,E2 -24151.907} C_VEL
LIN {X 0,Y 206.954,Z 530.961,A -85,B 0,C 180,E1 -24151.252,E2 -24151.252} C_VEL
LIN {X 0,Y 205.772,Z 534.754,A -85,B 0,C 180,E1 -24151.325,E2 -24151.325} C_VEL
LIN {X 0,Y 201.79,Z 550.135,A -85,B 0,C 180,E1 -24152.373,E2 -24152.373} C_VEL
LIN {X 0,Y 197.359,Z 564.397,A -85,B 0,C 180,E1 -24153.655,E2 -24153.655} C_VEL
LIN {X 0,Y 192.473,Z 577.953,A -85,B 0,C 180,E1 -24155.214,E2 -24155.214} C_VEL
LIN {X 0,Y 186.511,Z 592.079,A -85,B 0,C 180,E1 -24157.261,E2 -24157.261} C_VEL
LIN {X 0,Y 180.349,Z 605.184,A -85,B 0,C 180,E1 -24159.679,E2 -24159.679} C_VEL
LIN {X 0,Y 173.992,Z 617.445,A -85,B 0,C 180,E1 -24162.51,E2 -24162.51} C_VEL
LIN {X 0,Y 167.116,Z 629.6,A -85,B 0,C 180,E1 -24166.061,E2 -24166.061} C_VEL
LIN {X 0,Y 160.924,Z 639.863,A -85,B 0,C 180,E1 -24169.897,E2 -24169.897} C_VEL
LIN {X 0,Y 155.446,Z 648.663,A -85,B 0,C 180,E1 -24174.003,E2 -24174.003} C_VEL
LIN {X 0,Y 150.282,Z 657.205,A -85,B 0,C 180,E1 -24179.042,E2 -24179.042} C_VEL
LIN {X 0,Y 146.161,Z 664.235,A -85,B 0,C 180,E1 -24184.358,E2 -24184.358} C_VEL
LIN {X 0,Y 143.255,Z 669.961,A -85,B 0,C 180,E1 -24189.915,E2 -24189.915} C_VEL
LIN {X 0,Y 141.373,Z 674.557,A -85,B 0,C 180,E1 -24195.608,E2 -24195.608} C_VEL
LIN {X 0,Y 140.575,Z 677.95,A -85,B 0,C 180,E1 -24201.374,E2 -24201.374} C_VEL
LIN {X 0,Y 140.542,Z 680.352,A -85,B 0,C 180,E1 -24207.134,E2 -24207.134} C_VEL
LIN {X 0,Y 140.583,Z 681.376,A -85,B 0,C 180,E1 -24211.109,E2 -24211.109} C_VEL
LIN {X 0,Y 140.44,Z 681.94,A -85,B 0,C 180,E1 -24215.744,E2 -24215.744} C_VEL
LIN {X 0,Y 140.886,Z 681.817,A -85,B 0,C 180,E1 -24221.51,E2 -24221.51} C_VEL
LIN {X 0,Y 142.353,Z 680.724,A -85,B 0,C 180,E1 -24227.231,E2 -24227.231} C_VEL
LIN {X 0,Y 145.09,Z 678.628,A -85,B 0,C 180,E1 -24233.028,E2 -24233.028} C_VEL
LIN {X 0,Y 148.853,Z 675.735,A -85,B 0,C 180,E1 -24238.174,E2 -24238.174} C_VEL
LIN {X 0,Y 153.858,Z 671.767,A -85,B 0,C 180,E1 -24243.24,E2 -24243.24} C_VEL
LIN {X 0,Y 159.951,Z 666.718,A -85,B 0,C 180,E1 -24247.963,E2 -24247.963} C_VEL
LIN {X 0,Y 167.123,Z 660.586,A -85,B 0,C 180,E1 -24252.288,E2 -24252.288} C_VEL
LIN {X 0,Y 176.233,Z 652.109,A -85,B 0,C 180,E1 -24256.702,E2 -24256.702} C_VEL
LIN {X 0,Y 185.091,Z 643.046,A -85,B 0,C 180,E1 -24260.256,E2 -24260.256} C_VEL
LIN {X 0,Y 194.652,Z 632.322,A -85,B 0,C 180,E1 -24263.451,E2 -24263.451} C_VEL
LIN {X 0,Y 203.597,Z 621.293,A -85,B 0,C 180,E1 -24265.941,E2 -24265.941} C_VEL
LIN {X 0,Y 211.937,Z 609.598,A -85,B 0,C 180,E1 -24268.05,E2 -24268.05} C_VEL
LIN {X 0,Y 220.361,Z 596.279,A -85,B 0,C 180,E1 -24269.895,E2 -24269.895} C_VEL
LIN {X 0,Y 228.121,Z 582.176,A -85,B 0,C 180,E1 -24271.406,E2 -24271.406} C_VEL
LIN {X 0,Y 235.25,Z 566.802,A -85,B 0,C 180,E1 -24272.72,E2 -24272.72} C_VEL
LIN {X 0,Y 241.128,Z 551.814,A -85,B 0,C 180,E1 -24273.67,E2 -24273.67} C_VEL
LIN {X 0,Y 246.116,Z 535.823,A -85,B 0,C 180,E1 -24274.449,E2 -24274.449} C_VEL
LIN {X 0,Y 249.683,Z 521.078,A -85,B 0,C 180,E1 -24274.958,E2 -24274.958} C_VEL
LIN {X 0,Y 252.59,Z 503.531,A -85,B 0,C 180,E1 -24275.449,E2 -24275.449} C_VEL
LIN {X 0,Y 258.6,Z 444.093,A -85,B 0,C 180,E1 -24276.739,E2 -24276.739} C_VEL
LIN {X 0,Y 255.553,Z 436.343,A -85,B 0,C 180,E1 -24279.91,E2 -24279.91} C_VEL
LIN {X 0,Y 253.601,Z 432.628,A -85,B 0,C 180,E1 -24282.252,E2 -24282.252} C_VEL
LIN {X 0,Y 252.158,Z 429.702,A -85,B 0,C 180,E1 -24284.438,E2 -24284.438} C_VEL
LIN {X 0,Y 250.598,Z 426.385,A -85,B 0,C 180,E1 -24287.691,E2 -24287.691} C_VEL
LIN {X 0,Y 249.405,Z 424.27,A -85,B 0,C 180,E1 -24293.529,E2 -24293.529} C_VEL
LIN {X 0,Y 249.979,Z 425.263,A -85,B 0,C 180,E1 -24297.86,E2 -24297.86} C_VEL
LIN {X 0,Y 250.847,Z 426.577,A -85,B 0,C 180,E1 -24300.302,E2 -24300.302} C_VEL
LIN {X 0,Y 252.6,Z 430.379,A -85,B 0,C 180,E1 -24303.695,E2 -24303.695} C_VEL
LIN {X 0,Y 254.578,Z 434.393,A -85,B 0,C 180,E1 -24306.409,E2 -24306.409} C_VEL
LIN {X 0,Y 256.972,Z 439.192,A -85,B 0,C 180,E1 -24309.019,E2 -24309.019} C_VEL
LIN {X 0,Y 258.67,Z 442.866,A -85,B 0,C 180,E1 -24310.64,E2 -24310.64} C_VEL
LIN {X 0,Y 252.688,Z 501.492,A -85,B 0,C 180,E1 -24311.927,E2 -24311.927} C_VEL
LIN {X 0,Y 249.601,Z 518.482,A -85,B 0,C 180,E1 -24312.393,E2 -24312.393} C_VEL
LIN {X 0,Y 246.148,Z 532.649,A -85,B 0,C 180,E1 -24313.008,E2 -24313.008} C_VEL
LIN {X 0,Y 241.154,Z 548.601,A -85,B 0,C 180,E1 -24313.898,E2 -24313.898} C_VEL
LIN {X 0,Y 235.502,Z 563.137,A -85,B 0,C 180,E1 -24314.948,E2 -24314.948} C_VEL
LIN {X 0,Y 228.825,Z 577.424,A -85,B 0,C 180,E1 -24316.25,E2 -24316.25} C_VEL
LIN {X 0,Y 221.452,Z 590.961,A -85,B 0,C 180,E1 -24317.809,E2 -24317.809} C_VEL
LIN {X 0,Y 213.613,Z 603.552,A -85,B 0,C 180,E1 -24319.647,E2 -24319.647} C_VEL
LIN {X 0,Y 204.606,Z 616.128,A -85,B 0,C 180,E1 -24321.963,E2 -24321.963} C_VEL
LIN {X 0,Y 195.356,Z 627.538,A -85,B 0,C 180,E1 -24324.717,E2 -24324.717} C_VEL
LIN {X 0,Y 186.569,Z 637.208,A -85,B 0,C 180,E1 -24327.718,E2 -24327.718} C_VEL
LIN {X 0,Y 177.031,Z 646.675,A -85,B 0,C 180,E1 -24331.567,E2 -24331.567} C_VEL
LIN {X 0,Y 168.662,Z 654.253,A -85,B 0,C 180,E1 -24335.689,E2 -24335.689} C_VEL
LIN {X 0,Y 161.222,Z 660.478,A -85,B 0,C 180,E1 -24340.284,E2 -24340.284} C_VEL
LIN {X 0,Y 154.749,Z 665.418,A -85,B 0,C 180,E1 -24345.255,E2 -24345.255} C_VEL
LIN {X 0,Y 150.655,Z 668.366,A -85,B 0,C 180,E1 -24349.224,E2 -24349.224} C_VEL
LIN {X 0,Y 146.28,Z 671.295,A -85,B 0,C 180,E1 -24354.792,E2 -24354.792} C_VEL
LIN {X 0,Y 143.14,Z 673.168,A -85,B 0,C 180,E1 -24360.594,E2 -24360.594} C_VEL
LIN {X 0,Y 141.187,Z 673.955,A -85,B 0,C 180,E1 -24366.532,E2 -24366.532} C_VEL
LIN {X 0,Y 140.363,Z 673.8,A -85,B 0,C 180,E1 -24372.517,E2 -24372.517} C_VEL
LIN {X 0,Y 140.104,Z 672.575,A -85,B 0,C 180,E1 -24378.425,E2 -24378.425} C_VEL
LIN {X 0,Y 140.689,Z 670.452,A -85,B 0,C 180,E1 -24384.266,E2 -24384.266} C_VEL
LIN {X 0,Y 141.689,Z 667.264,A -85,B 0,C 180,E1 -24390,E2 -24390} C_VEL
LIN {X 0,Y 143.528,Z 663.111,A -85,B 0,C 180,E1 -24395.62,E2 -24395.62} C_VEL
LIN {X 0,Y 146.274,Z 657.833,A -85,B 0,C 180,E1 -24401.08,E2 -24401.08} C_VEL
LIN {X 0,Y 150.231,Z 651.346,A -85,B 0,C 180,E1 -24406.301,E2 -24406.301} C_VEL
LIN {X 0,Y 155.235,Z 643.571,A -85,B 0,C 180,E1 -24411.234,E2 -24411.234} C_VEL
LIN {X 0,Y 161.221,Z 634.241,A -85,B 0,C 180,E1 -24415.844,E2 -24415.844} C_VEL
LIN {X 0,Y 168.002,Z 623.114,A -85,B 0,C 180,E1 -24420.132,E2 -24420.132} C_VEL
LIN {X 0,Y 174.527,Z 611.593,A -85,B 0,C 180,E1 -24423.621,E2 -24423.621} C_VEL
LIN {X 0,Y 181.028,Z 599.047,A -85,B 0,C 180,E1 -24426.648,E2 -24426.648} C_VEL
LIN {X 0,Y 186.866,Z 586.657,A -85,B 0,C 180,E1 -24429.047,E2 -24429.047} C_VEL
LIN {X 0,Y 193.031,Z 571.885,A -85,B 0,C 180,E1 -24431.293,E2 -24431.293} C_VEL
LIN {X 0,Y 198.114,Z 557.287,A -85,B 0,C 180,E1 -24433.069,E2 -24433.069} C_VEL
LIN {X 0,Y 202.557,Z 542.436,A -85,B 0,C 180,E1 -24434.462,E2 -24434.462} C_VEL
LIN {X 0,Y 206.518,Z 526.149,A -85,B 0,C 180,E1 -24435.614,E2 -24435.614} C_VEL
LIN {X 0,Y 209.478,Z 510.283,A -85,B 0,C 180,E1 -24436.425,E2 -24436.425} C_VEL
LIN {X 0,Y 211.607,Z 493.167,A -85,B 0,C 180,E1 -24436.993,E2 -24436.993} C_VEL
LIN {X 0,Y 218.18,Z 413.622,A -85,B 0,C 180,E1 -24439.113,E2 -24439.113} C_VEL
LIN {X 0,Y 212.919,Z 402.892,A -85,B 0,C 180,E1 -24442.026,E2 -24442.026} C_VEL
LIN {X 0,Y 207.342,Z 392.706,A -85,B 0,C 180,E1 -24445.506,E2 -24445.506} C_VEL
LIN {X 0,Y 201.981,Z 383.698,A -85,B 0,C 180,E1 -24449.426,E2 -24449.426} C_VEL
LIN {X 0,Y 198.338,Z 378.039,A -85,B 0,C 180,E1 -24452.57,E2 -24452.57} C_VEL
LIN {X 0,Y 195.78,Z 374.254,A -85,B 0,C 180,E1 -24455.154,E2 -24455.154} C_VEL
LIN {X 0,Y 192.941,Z 369.995,A -85,B 0,C 180,E1 -24458.637,E2 -24458.637} C_VEL
LIN {X 0,Y 190.557,Z 366.769,A -85,B 0,C 180,E1 -24462.396,E2 -24462.396} C_VEL
LIN {X 0,Y 189.872,Z 365.337,A -85,B 0,C 180,E1 -24463.881,E2 -24463.881} C_VEL
LIN {X 0,Y 187.784,Z 362.85,A -85,B 0,C 180,E1 -24471.389,E2 -24471.389} C_VEL
LIN {X 0,Y 187.747,Z 362.757,A -85,B 0,C 180,E1 -24474.707,E2 -24474.707} C_VEL
LIN {X 0,Y 188.381,Z 363.397,A -85,B 0,C 180,E1 -24478.573,E2 -24478.573} C_VEL
LIN {X 0,Y 190.398,Z 365.709,A -85,B 0,C 180,E1 -24483.736,E2 -24483.736} C_VEL
LIN {X 0,Y 192.698,Z 369.543,A -85,B 0,C 180,E1 -24487.629,E2 -24487.629} C_VEL
LIN {X 0,Y 193.55,Z 370.719,A -85,B 0,C 180,E1 -24488.774,E2 -24488.774} C_VEL
LIN {X 0,Y 196.511,Z 375.237,A -85,B 0,C 180,E1 -24492.226,E2 -24492.226} C_VEL
LIN {X 0,Y 199.574,Z 379.931,A -85,B 0,C 180,E1 -24495.166,E2 -24495.166} C_VEL
LIN {X 0,Y 203.31,Z 385.727,A -85,B 0,C 180,E1 -24498.214,E2 -24498.214} C_VEL
LIN {X 0,Y 208.147,Z 394.128,A -85,B 0,C 180,E1 -24501.639,E2 -24501.639} C_VEL
LIN {X 0,Y 212.342,Z 401.782,A -85,B 0,C 180,E1 -24504.25,E2 -24504.25} C_VEL
LIN {X 0,Y 216.234,Z 411.264,A -85,B 0,C 180,E1 -24506.566,E2 -24506.566} C_VEL
LIN {X 0,Y 218.147,Z 416.301,A -85,B 0,C 180,E1 -24507.646,E2 -24507.646} C_VEL
LIN {X 0,Y 210.411,Z 507.87,A -85,B 0,C 180,E1 -24510.097,E2 -24510.097} C_VEL
LIN {X 0,Y 207.813,Z 524.545,A -85,B 0,C 180,E1 -24510.766,E2 -24510.766} C_VEL
LIN {X 0,Y 205.772,Z 534.754,A -85,B 0,C 180,E1 -24511.325,E2 -24511.325} C_VEL
LIN {X 0,Y 204.147,Z 540.377,A -85,B 0,C 180,E1 -24511.531,E2 -24511.531} C_VEL
LIN {X 0,Y 200.028,Z 549.388,A -85,B 0,C 180,E1 -24511.527,E2 -24511.527} C_VEL
LIN {X 0,Y 195.478,Z 558.2,A -85,B 0,C 180,E1 -24511.606,E2 -24511.606} C_VEL
LIN {X 0,Y 193.186,Z 563.514,A -85,B 0,C 180,E1 -24511.958,E2 -24511.958} C_VEL
LIN {X 0,Y 188.414,Z 576.459,A -85,B 0,C 180,E1 -24513.425,E2 -24513.425} C_VEL
LIN {X 0,Y 182.147,Z 590.965,A -85,B 0,C 180,E1 -24515.472,E2 -24515.472} C_VEL
LIN {X 0,Y 175.248,Z 605.195,A -85,B 0,C 180,E1 -24518.092,E2 -24518.092} C_VEL
LIN {X 0,Y 169.165,Z 616.502,A -85,B 0,C 180,E1 -24520.694,E2 -24520.694} C_VEL
LIN {X 0,Y 161.712,Z 629.182,A -85,B 0,C 180,E1 -24524.426,E2 -24524.426} C_VEL
LIN {X 0,Y 154.586,Z 640.488,A -85,B 0,C 180,E1 -24528.76,E2 -24528.76} C_VEL
LIN {X 0,Y 148.377,Z 649.946,A -85,B 0,C 180,E1 -24533.441,E2 -24533.441} C_VEL
LIN {X 0,Y 142.901,Z 658.489,A -85,B 0,C 180,E1 -24538.909,E2 -24538.909} C_VEL
LIN {X 0,Y 138.749,Z 665.292,A -85,B 0,C 180,E1 -24544.498,E2 -24544.498} C_VEL
LIN {X 0,Y 135.874,Z 670.78,A -85,B 0,C 180,E1 -24550.354,E2 -24550.354} C_VEL
LIN {X 0,Y 134.428,Z 674.157,A -85,B 0,C 180,E1 -24554.847,E2 -24554.847} C_VEL
LIN {X 0,Y 133.506,Z 677.601,A -85,B 0,C 180,E1 -24560.914,E2 -24560.914} C_VEL
LIN {X 0,Y 133.459,Z 680.068,A -85,B 0,C 180,E1 -24566.982,E2 -24566.982} C_VEL
LIN {X 0,Y 133.53,Z 680.938,A -85,B 0,C 180,E1 -24570.305,E2 -24570.305} C_VEL
LIN {X 0,Y 133.368,Z 681.716,A -85,B 0,C 180,E1 -24576.05,E2 -24576.05} C_VEL
LIN {X 0,Y 133.866,Z 681.623,A -85,B 0,C 180,E1 -24582.123,E2 -24582.123} C_VEL
LIN {X 0,Y 135.519,Z 680.595,A -85,B 0,C 180,E1 -24588.129,E2 -24588.129} C_VEL
LIN {X 0,Y 138.362,Z 678.619,A -85,B 0,C 180,E1 -24593.976,E2 -24593.976} C_VEL
LIN {X 0,Y 142.563,Z 675.705,A -85,B 0,C 180,E1 -24599.537,E2 -24599.537} C_VEL
LIN {X 0,Y 147.899,Z 671.771,A -85,B 0,C 180,E1 -24604.766,E2 -24604.766} C_VEL
LIN {X 0,Y 154.351,Z 666.795,A -85,B 0,C 180,E1 -24609.603,E2 -24609.603} C_VEL
LIN {X 0,Y 161.882,Z 660.7,A -85,B 0,C 180,E1 -24613.998,E2 -24613.998} C_VEL
LIN {X 0,Y 171.397,Z 652.304,A -85,B 0,C 180,E1 -24618.446,E2 -24618.446} C_VEL
LIN {X 0,Y 180.617,Z 643.329,A -85,B 0,C 180,E1 -24621.995,E2 -24621.995} C_VEL
LIN {X 0,Y 190.51,Z 632.705,A -85,B 0,C 180,E1 -24625.167,E2 -24625.167} C_VEL
LIN {X 0,Y 199.716,Z 621.793,A -85,B 0,C 180,E1 -24627.625,E2 -24627.625} C_VEL
LIN {X 0,Y 208.273,Z 610.168,A -85,B 0,C 180,E1 -24629.705,E2 -24629.705} C_VEL
LIN {X 0,Y 216.912,Z 597.024,A -85,B 0,C 180,E1 -24631.506,E2 -24631.506} C_VEL
LIN {X 0,Y 224.847,Z 583.144,A -85,B 0,C 180,E1 -24632.977,E2 -24632.977} C_VEL
LIN {X 0,Y 232.131,Z 568.063,A -85,B 0,C 180,E1 -24634.252,E2 -24634.252} C_VEL
LIN {X 0,Y 238.482,Z 552.342,A -85,B 0,C 180,E1 -24635.236,E2 -24635.236} C_VEL
LIN {X 0,Y 243.375,Z 537.147,A -85,B 0,C 180,E1 -24635.958,E2 -24635.958} C_VEL
LIN {X 0,Y 247.337,Z 521.409,A -85,B 0,C 180,E1 -24636.501,E2 -24636.501} C_VEL
LIN {X 0,Y 250.196,Z 505.19,A -85,B 0,C 180,E1 -24636.944,E2 -24636.944} C_VEL
LIN {X 0,Y 256.121,Z 448.675,A -85,B 0,C 180,E1 -24638.133,E2 -24638.133} C_VEL
LIN {X 0,Y 255.942,Z 447.836,A -85,B 0,C 180,E1 -24638.357,E2 -24638.357} C_VEL
LIN {X 0,Y 253.981,Z 442.62,A -85,B 0,C 180,E1 -24640.607,E2 -24640.607} C_VEL
LIN {X 0,Y 252.175,Z 438.993,A -85,B 0,C 180,E1 -24642.941,E2 -24642.941} C_VEL
LIN {X 0,Y 250.943,Z 436.385,A -85,B 0,C 180,E1 -24644.956,E2 -24644.956} C_VEL
LIN {X 0,Y 249.531,Z 433.303,A -85,B 0,C 180,E1 -24648.134,E2 -24648.134} C_VEL
LIN {X 0,Y 248.529,Z 431.325,A -85,B 0,C 180,E1 -24653.506,E2 -24653.506} C_VEL
LIN {X 0,Y 249.095,Z 432.336,A -85,B 0,C 180,E1 -24657.853,E2 -24657.853} C_VEL
LIN {X 0,Y 249.832,Z 433.476,A -85,B 0,C 180,E1 -24660.001,E2 -24660.001} C_VEL
LIN {X 0,Y 251.47,Z 437.268,A -85,B 0,C 180,E1 -24663.364,E2 -24663.364} C_VEL
LIN {X 0,Y 253.203,Z 440.938,A -85,B 0,C 180,E1 -24665.875,E2 -24665.875} C_VEL
LIN {X 0,Y 255.556,Z 445.933,A -85,B 0,C 180,E1 -24668.579,E2 -24668.579} C_VEL
LIN {X 0,Y 256.187,Z 447.363,A -85,B 0,C 180,E1 -24669.23,E2 -24669.23} C_VEL
LIN {X 0,Y 250.356,Z 502.683,A -85,B 0,C 180,E1 -24670.42,E2 -24670.42} C_VEL
LIN {X 0,Y 247.125,Z 519.719,A -85,B 0,C 180,E1 -24670.875,E2 -24670.875} C_VEL
LIN {X 0,Y 243.462,Z 534.113,A -85,B 0,C 180,E1 -24671.508,E2 -24671.508} C_VEL
LIN {X 0,Y 238.633,Z 549.026,A -85,B 0,C 180,E1 -24672.316,E2 -24672.316} C_VEL
LIN {X 0,Y 232.928,Z 563.383,A -85,B 0,C 180,E1 -24673.328,E2 -24673.328} C_VEL
LIN {X 0,Y 225.965,Z 577.913,A -85,B 0,C 180,E1 -24674.618,E2 -24674.618} C_VEL
LIN {X 0,Y 218.539,Z 591.162,A -85,B 0,C 180,E1 -24676.105,E2 -24676.105} C_VEL
LIN {X 0,Y 210.436,Z 603.78,A -85,B 0,C 180,E1 -24677.894,E2 -24677.894} C_VEL
LIN {X 0,Y 201.12,Z 616.442,A -85,B 0,C 180,E1 -24680.2,E2 -24680.2} C_VEL
LIN {X 0,Y 190.998,Z 628.493,A -85,B 0,C 180,E1 -24683.087,E2 -24683.087} C_VEL
LIN {X 0,Y 181.909,Z 638.033,A -85,B 0,C 180,E1 -24686.07,E2 -24686.07} C_VEL
LIN {X 0,Y 172.763,Z 646.729,A -85,B 0,C 180,E1 -24689.619,E2 -24689.619} C_VEL
LIN {X 0,Y 163.497,Z 654.695,A -85,B 0,C 180,E1 -24693.975,E2 -24693.975} C_VEL
LIN {X 0,Y 154.578,Z 661.703,A -85,B 0,C 180,E1 -24699.383,E2 -24699.383} C_VEL
LIN {X 0,Y 147.898,Z 666.435,A -85,B 0,C 180,E1 -24704.537,E2 -24704.537} C_VEL
LIN {X 0,Y 142.416,Z 669.982,A -85,B 0,C 180,E1 -24710.094,E2 -24710.094} C_VEL
LIN {X 0,Y 138.231,Z 672.482,A -85,B 0,C 180,E1 -24715.994,E2 -24715.994} C_VEL
LIN {X 0,Y 135.363,Z 673.832,A -85,B 0,C 180,E1 -24722.142,E2 -24722.142} C_VEL
LIN {X 0,Y 133.705,Z 674.237,A -85,B 0,C 180,E1 -24728.411,E2 -24728.411} C_VEL
LIN {X 0,Y 133.351,Z 674.037,A -85,B 0,C 180,E1 -24731.565,E2 -24731.565} C_VEL
LIN {X 0,Y 132.987,Z 672.893,A -85,B 0,C 180,E1 -24737.796,E2 -24737.796} C_VEL
LIN {X 0,Y 133.524,Z 670.832,A -85,B 0,C 180,E1 -24743.957,E2 -24743.957} C_VEL
LIN {X 0,Y 134.026,Z 669.379,A -85,B 0,C 180,E1 -24746.994,E2 -24746.994} C_VEL
LIN {X 0,Y 135.939,Z 664.727,A -85,B 0,C 180,E1 -24754.447,E2 -24754.447} C_VEL
LIN {X 0,Y 138.516,Z 659.821,A -85,B 0,C 180,E1 -24760.229,E2 -24760.229} C_VEL
LIN {X 0,Y 142.322,Z 653.756,A -85,B 0,C 180,E1 -24765.759,E2 -24765.759} C_VEL
LIN {X 0,Y 147.962,Z 645.346,A -85,B 0,C 180,E1 -24771.599,E2 -24771.599} C_VEL
LIN {X 0,Y 154.033,Z 636.3,A -85,B 0,C 180,E1 -24776.414,E2 -24776.414} C_VEL
LIN {X 0,Y 161.049,Z 625.54,A -85,B 0,C 180,E1 -24780.847,E2 -24780.847} C_VEL
LIN {X 0,Y 167.721,Z 614.463,A -85,B 0,C 180,E1 -24784.45,E2 -24784.45} C_VEL
LIN {X 0,Y 173.821,Z 603.392,A -85,B 0,C 180,E1 -24787.336,E2 -24787.336} C_VEL
LIN {X 0,Y 180.303,Z 590.429,A -85,B 0,C 180,E1 -24790.027,E2 -24790.027} C_VEL
LIN {X 0,Y 186.643,Z 576.352,A -85,B 0,C 180,E1 -24792.305,E2 -24792.305} C_VEL
LIN {X 0,Y 191.895,Z 562.742,A -85,B 0,C 180,E1 -24794.096,E2 -24794.096} C_VEL
LIN {X 0,Y 196.973,Z 547.071,A -85,B 0,C 180,E1 -24795.711,E2 -24795.711} C_VEL
LIN {X 0,Y 201.402,Z 530.588,A -85,B 0,C 180,E1 -24796.938,E2 -24796.938} C_VEL
LIN {X 0,Y 204.709,Z 514.213,A -85,B 0,C 180,E1 -24797.846,E2 -24797.846} C_VEL
LIN {X 0,Y 207.119,Z 497.36,A -85,B 0,C 180,E1 -24798.467,E2 -24798.467} C_VEL
LIN {X 0,Y 214.064,Z 416.694,A -85,B 0,C 180,E1 -24800.628,E2 -24800.628} C_VEL
LIN {X 0,Y 209.312,Z 406.837,A -85,B 0,C 180,E1 -24803.469,E2 -24803.469} C_VEL
LIN {X 0,Y 204.556,Z 397.966,A -85,B 0,C 180,E1 -24806.651,E2 -24806.651} C_VEL
LIN {X 0,Y 199.577,Z 389.238,A -85,B 0,C 180,E1 -24810.548,E2 -24810.548} C_VEL
LIN {X 0,Y 196.268,Z 384.023,A -85,B 0,C 180,E1 -24813.605,E2 -24813.605} C_VEL
LIN {X 0,Y 194.193,Z 380.805,A -85,B 0,C 180,E1 -24815.845,E2 -24815.845} C_VEL
LIN {X 0,Y 191.549,Z 376.709,A -85,B 0,C 180,E1 -24819.273,E2 -24819.273} C_VEL
LIN {X 0,Y 189.264,Z 373.277,A -85,B 0,C 180,E1 -24823.178,E2 -24823.178} C_VEL
LIN {X 0,Y 188.874,Z 372.336,A -85,B 0,C 180,E1 -24824.1,E2 -24824.1} C_VEL
LIN {X 0,Y 186.841,Z 369.782,A -85,B 0,C 180,E1 -24832.458,E2 -24832.458} C_VEL
LIN {X 0,Y 187.328,Z 370.248,A -85,B 0,C 180,E1 -24837.849,E2 -24837.849} C_VEL
LIN {X 0,Y 189.249,Z 372.564,A -85,B 0,C 180,E1 -24843.253,E2 -24843.253} C_VEL
LIN {X 0,Y 191.567,Z 376.482,A -85,B 0,C 180,E1 -24847.334,E2 -24847.334} C_VEL
LIN {X 0,Y 192.437,Z 377.937,A -85,B 0,C 180,E1 -24848.569,E2 -24848.569} C_VEL
LIN {X 0,Y 195.069,Z 382.012,A -85,B 0,C 180,E1 -24851.733,E2 -24851.733} C_VEL
LIN {X 0,Y 197.716,Z 386.284,A -85,B 0,C 180,E1 -24854.407,E2 -24854.407} C_VEL
LIN {X 0,Y 201.19,Z 391.872,A -85,B 0,C 180,E1 -24857.395,E2 -24857.395} C_VEL
LIN {X 0,Y 205.681,Z 399.919,A -85,B 0,C 180,E1 -24860.742,E2 -24860.742} C_VEL
LIN {X 0,Y 209.555,Z 407.337,A -85,B 0,C 180,E1 -24863.301,E2 -24863.301} C_VEL
LIN {X 0,Y 213.522,Z 417.505,A -85,B 0,C 180,E1 -24865.803,E2 -24865.803} C_VEL
LIN {X 0,Y 214.079,Z 418.976,A -85,B 0,C 180,E1 -24866.135,E2 -24866.135} C_VEL
LIN {X 0,Y 206.301,Z 507.991,A -85,B 0,C 180,E1 -24868.508,E2 -24868.508} C_VEL
LIN {X 0,Y 203.657,Z 524.43,A -85,B 0,C 180,E1 -24869.164,E2 -24869.164} C_VEL
LIN {X 0,Y 200.019,Z 540.713,A -85,B 0,C 180,E1 -24870.09,E2 -24870.09} C_VEL
LIN {X 0,Y 195.399,Z 556.794,A -85,B 0,C 180,E1 -24871.326,E2 -24871.326} C_VEL
LIN {X 0,Y 193.186,Z 563.514,A -85,B 0,C 180,E1 -24871.958,E2 -24871.958} C_VEL
LIN {X 0,Y 190.808,Z 568.918,A -85,B 0,C 180,E1 -24872.351,E2 -24872.351} C_VEL
LIN {X 0,Y 181.341,Z 583.902,A -85,B 0,C 180,E1 -24872.949,E2 -24872.949} C_VEL
LIN {X 0,Y 178.492,Z 588.806,A -85,B 0,C 180,E1 -24873.439,E2 -24873.439} C_VEL
LIN {X 0,Y 177.704,Z 590.398,A -85,B 0,C 180,E1 -24873.681,E2 -24873.681} C_VEL
LIN {X 0,Y 170.902,Z 604.118,A -85,B 0,C 180,E1 -24876.193,E2 -24876.193} C_VEL
LIN {X 0,Y 164.514,Z 615.516,A -85,B 0,C 180,E1 -24878.773,E2 -24878.773} C_VEL
LIN {X 0,Y 157.348,Z 627.27,A -85,B 0,C 180,E1 -24882.193,E2 -24882.193} C_VEL
LIN {X 0,Y 150.124,Z 638.334,A -85,B 0,C 180,E1 -24886.329,E2 -24886.329} C_VEL
LIN {X 0,Y 143.216,Z 648.387,A -85,B 0,C 180,E1 -24891.198,E2 -24891.198} C_VEL
LIN {X 0,Y 138.044,Z 656.023,A -85,B 0,C 180,E1 -24895.943,E2 -24895.943} C_VEL
LIN {X 0,Y 133.252,Z 663.165,A -85,B 0,C 180,E1 -24901.662,E2 -24901.662} C_VEL
LIN {X 0,Y 129.779,Z 669.044,A -85,B 0,C 180,E1 -24907.724,E2 -24907.724} C_VEL
LIN {X 0,Y 127.515,Z 673.733,A -85,B 0,C 180,E1 -24914.004,E2 -24914.004} C_VEL
LIN {X 0,Y 126.461,Z 677.248,A -85,B 0,C 180,E1 -24920.403,E2 -24920.403} C_VEL
LIN {X 0,Y 126.367,Z 679.766,A -85,B 0,C 180,E1 -24926.812,E2 -24926.812} C_VEL
LIN {X 0,Y 126.466,Z 680.574,A -85,B 0,C 180,E1 -24930,E2 -24930} C_VEL
LIN {X 0,Y 126.27,Z 681.492,A -85,B 0,C 180,E1 -24936.392,E2 -24936.392} C_VEL
LIN {X 0,Y 126.874,Z 681.43,A -85,B 0,C 180,E1 -24942.802,E2 -24942.802} C_VEL
LIN {X 0,Y 128.728,Z 680.465,A -85,B 0,C 180,E1 -24949.122,E2 -24949.122} C_VEL
LIN {X 0,Y 131.827,Z 678.521,A -85,B 0,C 180,E1 -24955.246,E2 -24955.246} C_VEL
LIN {X 0,Y 136.334,Z 675.674,A -85,B 0,C 180,E1 -24961.031,E2 -24961.031} C_VEL
LIN {X 0,Y 143.627,Z 670.69,A -85,B 0,C 180,E1 -24967.71,E2 -24967.71} C_VEL
LIN {X 0,Y 152.736,Z 664.019,A -85,B 0,C 180,E1 -24973.647,E2 -24973.647} C_VEL
LIN {X 0,Y 161.074,Z 657.315,A -85,B 0,C 180,E1 -24977.881,E2 -24977.881} C_VEL
LIN {X 0,Y 170.748,Z 648.854,A -85,B 0,C 180,E1 -24981.875,E2 -24981.875} C_VEL
LIN {X 0,Y 180.088,Z 639.918,A -85,B 0,C 180,E1 -24985.039,E2 -24985.039} C_VEL
LIN {X 0,Y 189.244,Z 630.151,A -85,B 0,C 180,E1 -24987.659,E2 -24987.659} C_VEL
LIN {X 0,Y 198.532,Z 619.061,A -85,B 0,C 180,E1 -24989.999,E2 -24989.999} C_VEL
LIN {X 0,Y 207.149,Z 607.558,A -85,B 0,C 180,E1 -24991.898,E2 -24991.898} C_VEL
LIN {X 0,Y 215.857,Z 594.318,A -85,B 0,C 180,E1 -24993.555,E2 -24993.555} C_VEL
LIN {X 0,Y 223.951,Z 579.917,A -85,B 0,C 180,E1 -24994.98,E2 -24994.98} C_VEL
LIN {X 0,Y 230.68,Z 565.852,A -85,B 0,C 180,E1 -24996.064,E2 -24996.064} C_VEL
LIN {X 0,Y 236.773,Z 550.723,A -85,B 0,C 180,E1 -24996.949,E2 -24996.949} C_VEL
LIN {X 0,Y 241.75,Z 535.281,A -85,B 0,C 180,E1 -24997.644,E2 -24997.644} C_VEL
LIN {X 0,Y 245.704,Z 519.267,A -85,B 0,C 180,E1 -24998.144,E2 -24998.144} C_VEL
LIN {X 0,Y 248.492,Z 502.618,A -85,B 0,C 180,E1 -24998.573,E2 -24998.573} C_VEL
LIN {X 0,Y 253.803,Z 452.636,A -85,B 0,C 180,E1 -24999.615,E2 -24999.615} C_VEL
LIN {X 0,Y 252.382,Z 448.677,A -85,B 0,C 180,E1 -25001.406,E2 -25001.406} C_VEL
LIN {X 0,Y 250.07,Z 443.606,A -85,B 0,C 180,E1 -25004.902,E2 -25004.902} C_VEL
LIN {X 0,Y 248.587,Z 440.305,A -85,B 0,C 180,E1 -25008.297,E2 -25008.297} C_VEL
LIN {X 0,Y 247.653,Z 438.381,A -85,B 0,C 180,E1 -25013.483,E2 -25013.483} C_VEL
LIN {X 0,Y 248.141,Z 439.302,A -85,B 0,C 180,E1 -25017.578,E2 -25017.578} C_VEL
LIN {X 0,Y 248.813,Z 440.379,A -85,B 0,C 180,E1 -25019.675,E2 -25019.675} C_VEL
LIN {X 0,Y 250.312,Z 444.053,A -85,B 0,C 180,E1 -25022.96,E2 -25022.96} C_VEL
LIN {X 0,Y 251.945,Z 447.708,A -85,B 0,C 180,E1 -25025.466,E2 -25025.466} C_VEL
LIN {X 0,Y 253.857,Z 451.924,A -85,B 0,C 180,E1 -25027.796,E2 -25027.796} C_VEL
LIN {X 0,Y 248.39,Z 502.491,A -85,B 0,C 180,E1 -25028.851,E2 -25028.851} C_VEL
LIN {X 0,Y 245.029,Z 520.009,A -85,B 0,C 180,E1 -25029.3,E2 -25029.3} C_VEL
LIN {X 0,Y 241.518,Z 533.556,A -85,B 0,C 180,E1 -25029.86,E2 -25029.86} C_VEL
LIN {X 0,Y 236.506,Z 548.908,A -85,B 0,C 180,E1 -25030.667,E2 -25030.667} C_VEL
LIN {X 0,Y 230.54,Z 563.626,A -85,B 0,C 180,E1 -25031.669,E2 -25031.669} C_VEL
LIN {X 0,Y 223.513,Z 577.985,A -85,B 0,C 180,E1 -25032.904,E2 -25032.904} C_VEL
LIN {X 0,Y 215.832,Z 591.394,A -85,B 0,C 180,E1 -25034.364,E2 -25034.364} C_VEL
LIN {X 0,Y 207.801,Z 603.621,A -85,B 0,C 180,E1 -25036.04,E2 -25036.04} C_VEL
LIN {X 0,Y 198.402,Z 616.042,A -85,B 0,C 180,E1 -25038.224,E2 -25038.224} C_VEL
LIN {X 0,Y 189.554,Z 626.373,A -85,B 0,C 180,E1 -25040.579,E2 -25040.579} C_VEL
LIN {X 0,Y 180.05,Z 636.308,A -85,B 0,C 180,E1 -25043.466,E2 -25043.466} C_VEL
LIN {X 0,Y 170.09,Z 645.622,A -85,B 0,C 180,E1 -25047.035,E2 -25047.035} C_VEL
LIN {X 0,Y 160.31,Z 653.742,A -85,B 0,C 180,E1 -25051.255,E2 -25051.255} C_VEL
LIN {X 0,Y 151.821,Z 660.139,A -85,B 0,C 180,E1 -25055.894,E2 -25055.894} C_VEL
LIN {X 0,Y 144.359,Z 665.277,A -85,B 0,C 180,E1 -25061.009,E2 -25061.009} C_VEL
LIN {X 0,Y 139.502,Z 668.32,A -85,B 0,C 180,E1 -25065.145,E2 -25065.145} C_VEL
LIN {X 0,Y 133.34,Z 671.861,A -85,B 0,C 180,E1 -25072.245,E2 -25072.245} C_VEL
LIN {X 0,Y 130.212,Z 673.39,A -85,B 0,C 180,E1 -25077.334,E2 -25077.334} C_VEL
LIN {X 0,Y 127.635,Z 674.347,A -85,B 0,C 180,E1 -25083.863,E2 -25083.863} C_VEL
LIN {X 0,Y 126.293,Z 674.239,A -85,B 0,C 180,E1 -25091.094,E2 -25091.094} C_VEL
LIN {X 0,Y 125.876,Z 673.21,A -85,B 0,C 180,E1 -25097.095,E2 -25097.095} C_VEL
LIN {X 0,Y 126.354,Z 671.187,A -85,B 0,C 180,E1 -25103.613,E2 -25103.613} C_VEL
LIN {X 0,Y 126.895,Z 669.773,A -85,B 0,C 180,E1 -25106.825,E2 -25106.825} C_VEL
LIN {X 0,Y 128.28,Z 666.276,A -85,B 0,C 180,E1 -25113.14,E2 -25113.14} C_VEL
LIN {X 0,Y 130.806,Z 661.688,A -85,B 0,C 180,E1 -25119.275,E2 -25119.275} C_VEL
LIN {X 0,Y 134.375,Z 655.979,A -85,B 0,C 180,E1 -25125.159,E2 -25125.159} C_VEL
LIN {X 0,Y 139.982,Z 648.068,A -85,B 0,C 180,E1 -25131.346,E2 -25131.346} C_VEL
LIN {X 0,Y 146.085,Z 639.564,A -85,B 0,C 180,E1 -25136.423,E2 -25136.423} C_VEL
LIN {X 0,Y 153.123,Z 629.359,A -85,B 0,C 180,E1 -25141.087,E2 -25141.087} C_VEL
LIN {X 0,Y 159.917,Z 618.833,A -85,B 0,C 180,E1 -25144.842,E2 -25144.842} C_VEL
LIN {X 0,Y 167.195,Z 606.516,A -85,B 0,C 180,E1 -25148.317,E2 -25148.317} C_VEL
LIN {X 0,Y 173.85,Z 594.138,A -85,B 0,C 180,E1 -25151.065,E2 -25151.065} C_VEL
LIN {X 0,Y 180.324,Z 580.723,A -85,B 0,C 180,E1 -25153.387,E2 -25153.387} C_VEL
